# B&R Automation Studio project NAINV104C00R8L515F00 (part 4)

#### Types.typ - Exported data types
```iecst
(*HermesState*)

TYPE
	eHermesState :
		(
		HermesStateNotConnected,
		HermesStateConnected,
		HermesStateServiceDescription,
		HermesStateSServiceDescription,
		HermesStateNotAvailableNotReady,
		HermesStateBoardAvailable,
		HermesStateMachineReady,
		HermesStateAvailableAndReady,
		HermesStateTransporting,
		HermesStateTransportStopped,
		HermesStateTransportFinished
		);
END_TYPE

(**)
(*Hermes Message Type*)

TYPE
	tyHermesMsgType : 	STRUCT
		bCheckAlive : BOOL; (*Check Alive*)
		bCheckAlivePing : BOOL; (*Check Alive Ping*)
		bCheckAlivePong : BOOL; (*Check Alive Pong*)
		bServiceDescription : BOOL; (*Service Description*)
		bSServiceDescription : BOOL; (*Supervisory Service Description*)
		bNotification : BOOL; (*Notification*)
		bBoardAvailable : BOOL; (*Board Available*)
		bRevokeBoardAvailable : BOOL; (*Revoke Board Available*)
		bMachineReady : BOOL; (*Machine Ready*)
		bRevokeMachineReady : BOOL; (*Revoke Machine Ready*)
		bStartTransport : BOOL; (*Start Transport*)
		bStopTransport : BOOL; (*Stop Transport*)
		bTransportFinished : BOOL; (*Transport Finished*)
		bSetConfiguration : BOOL; (*Set Configuration*)
		bGetConfiguration : BOOL; (*Get Configuration*)
		bCurrentConfiguration : BOOL; (*Current Configuration*)
		bBoardForecast : BOOL; (*Board Forecast*)
		bBoardArrived : BOOL; (*Board Arrived*)
		bBoardDeparted : BOOL; (*Board Departed*)
		bQueryBoardInfo : BOOL; (*Query Board Info*)
		bSendBoardInfo : BOOL; (*Send Board Info*)
		bQueryWorkOrderInfo : BOOL; (*Query Work Order*)
		bSendWorkOrderInfo : BOOL; (*Send Work Order*)
		bCommand : BOOL;
	END_STRUCT;
	eHermesMsgType :
		(
		HermesMsgTypeNA, (*NA*)
		HermesMsgTypeCheckAlive, (*Check Alive*)
		HermesMsgTypeCheckAlivePing, (*Check Alive Ping*)
		HermesMsgTypeCheckAlivePong, (*Check Alive Pong*)
		HermesMsgTypeServiceDescription, (*Service Description*)
		HermesMsgTypeSServiceDescription, (*Supervisory Service Description*)
		HermesMsgTypeNotification, (*Notification*)
		HermesMsgTypeBoardAvailable, (*Board Available*)
		HermesMsgTypeRevokeBoardAvl, (*Revoke Board Available*)
		HermesMsgTypeMachineReady, (*Machine Ready*)
		HermesMsgTypeRevokeMachineReady, (*Revoke Machine Ready*)
		HermesMsgTypeStartTransport, (*Start Transport*)
		HermesMsgTypeStopTransport, (*Stop Transport*)
		HermesMsgTypeTransportFinished, (*Transport Finished*)
		HermesMsgTypeSetConfiguration, (*Set Configuration*)
		HermesMsgTypeGetConfiguration, (*Get Configuration*)
		HermesMsgTypeCurrConfiguration, (*Current Configuration*)
		HermesMsgTypeBoardForecast, (*Board Forecast*)
		HermesMsgTypeBoardForecastId, (*Board Forecast with Id*)
		HermesMsgTypeBoardForecastNoId, (*Board Forecast with no Id*)
		HermesMsgTypeBoardArrived, (*Board Arrived*)
		HermesMsgTypeBoardDeparted, (*Board Departed*)
		HermesMsgTypeQueryBoardInfo, (*Query Board Info*)
		HermesMsgTypeSendBoardInfo, (*Send Board Info*)
		HermesMsgTypeQueryWorkOrderInfo, (*Query Work Order Info*)
		HermesMsgTypeSendWorkOrderInfo, (*Send Work Order Info*)
		HermesMsgTypeCommand
		);
END_TYPE

(**)

TYPE
	eHermesCheckAliveType :
		(
		HermesCheckAliveTypeUnknown := 0, (*CheckAlive unknown*)
		HermesCheckAliveTypePing := 1, (*CheckAlive request*)
		HermesCheckAliveTypePong := 2 (*CheckAlive response*)
		);
	eHermesBoardTransfer :
		(
		HermesTransferred := 1, (*Transferred from upstream*)
		HermesLoaded := 2, (*Loaded from Magazine or a stack of Boards*)
		HermesInserted := 3 (*Inserted*)
		);
	eHermesFailedBoard :
		(
		HermesUnknownBoard := 0, (*Board of unknown quality available / Ready to accept any board*)
		HermesGoodBoard := 1, (*Good board available / Ready to accept good boards*)
		HermesFailedBoard := 2 (*Failed board available / Ready to accept failed boards*)
		);
	eHermesFlippedBoard :
		(
		HermesFlippedBoardUnknownSide := 0, (*Side up is unknown*)
		HermesFlippedBoardTopSideUp := 1, (*Board top side is up*)
		HermesFlippedBoardBtmSideUp := 2 (*Board bottom side is up*)
		);
	eHermesSeverity :
		(
		HermesSeverityFatalError := 1, (*Fatal Error*)
		HermesSeverityError := 2, (*Error*)
		HermesSeverityWarning := 3, (*Warning*)
		HermesSeverityInfo := 4 (*Info*)
		);
	eHermesTransferState :
		(
		HermesTransferStateNotStarted := 1, (*The PCB never left and hence is fully inside the upstream machine*)
		HermesTransferStateIncomplete := 2, (*The transfer was cancelled in progress*)
		HermesTransferStateComplete := 3 (*The transfer ended successfully*)
		);
END_TYPE

(**)
(**)
(*Command*)

TYPE
	tyHermesCmdProcessList : 	STRUCT
		bUSTrueDSFalse : BOOL;
		udiInterfaceString : UDINT;
		udiComMode : UDINT;
		udiCommandParam : UDINT;
	END_STRUCT;
	tyHermesCommandParam : 	STRUCT
		usiCommandIdx : USINT;
		eCommand : eHermesCommand;
		udiMsgCmdBffr : UDINT;
		a_eCommandSndQ : ARRAY[0..20]OF eHermesCommand;
	END_STRUCT;
	eHermesCommand :
		(
		HermesCommandUndefined := 0,
		HermesCommandLockInputConveyor := 1,
		HermesCommandUnLockInputConveyor := 2,
		HermesCommandRequestPause := 3,
		HermesCommandConfirmPause := 4,
		HermesCommandResumeOperation := 5,
		HermesCommandOvenInfeed := 1000,
		HermesCommandSelfDefine := 1001
		);
	tyHermesCommandPause : 	STRUCT
		bFeatureRequestTo : BOOL;
		bUnlockCoverSigTo : BOOL;
		bPrevUnlockCoverSigTo : BOOL;
		bMachineSafetySigFrom : BOOL;
		bFeatureRequestFrom : BOOL;
		bUnlockCoverSigFrom : BOOL;
		bMachineSafetySigTo : BOOL;
		bPrevMachineSafetySigTo : BOOL;
	END_STRUCT;
	tyHermesCommandLockConv : 	STRUCT
		bFeatureLockConvFrom : BOOL;
		bOvenInfoFrom : BOOL;
		bFeatureLockConvTo : BOOL;
		bOvenInfoTo : BOOL;
		bPrevOvenInfoTo : BOOL;
	END_STRUCT;
	tyHermesCommandOvenInfeed : 	STRUCT
		bFeatureOvenInfeedFrom : BOOL;
		bOvenInfeedFrom : BOOL;
		bFeatureOvenInfeedTo : BOOL;
		bOvenInfeedTo : BOOL;
		bPrevOvenInfeedTo : BOOL;
	END_STRUCT;
END_TYPE

(**)
(*Hermes Message Full Data*)

TYPE
	tyHermesNotification : 	STRUCT
		tyData : tyHermesNotificationData; (*Data*)
		tyAvl : tyHermesNotificationAvl; (*Availability*)
	END_STRUCT;
	tyHermesServiceDescription : 	STRUCT
		tyData : tyHermesServiceDescriptionData; (*Data*)
		tyAvl : tyHermesServiceDescriptionAvl; (*Availability*)
	END_STRUCT;
	tyHermesSServiceDescription : 	STRUCT
		tyData : tyHermesSServiceDescriptionData; (*Data*)
		tyAvl : tyHermesSServiceDescriptionAvl; (*Availability*)
	END_STRUCT;
	tyHermesCheckAlive : 	STRUCT
		tyData : tyHermesCheckAliveData; (*Data*)
		tyAvl : tyHermesCheckAliveAvl; (*Availability*)
	END_STRUCT;
	tyHermesBoardAvailable : 	STRUCT
		tyData : tyHermesBoardAvailableData; (*Data*)
		tyAvl : tyHermesBoardAvailableAvl; (*Availability*)
	END_STRUCT;
	tyHermesMachineReady : 	STRUCT
		tyData : tyHermesMachineReadyData; (*Data*)
		tyAvl : tyHermesMachineReadyAvl; (*Availability*)
	END_STRUCT;
	tyHermesStartTransport : 	STRUCT
		tyData : tyHermesStartTransportData; (*Data*)
		tyAvl : tyHermesStartTransportAvl; (*Availability*)
	END_STRUCT;
	tyHermesStopTransport : 	STRUCT
		tyData : tyHermesStopTransportData; (*Data*)
		tyAvl : tyHermesStopTransportAvl; (*Availability*)
	END_STRUCT;
	tyHermesTransportFinished : 	STRUCT
		tyData : tyHermesTransportFinishedData; (*Data*)
		tyAvl : tyHermesTransportFinishedAvl; (*Availability*)
	END_STRUCT;
	tyHermesBoardForecast : 	STRUCT
		tyData : tyHermesBoardForecastData; (*Data*)
		tyAvl : tyHermesBoardForecastAvl; (*Availability*)
	END_STRUCT;
	tyHermesQueryBoardInfo : 	STRUCT
		tyData : tyHermesQueryBoardInfoData; (*Data*)
		tyAvl : tyHermesQueryBoardInfoAvl; (*Availability*)
	END_STRUCT;
	tyHermesSendBoardInfo : 	STRUCT
		tyData : tyHermesSendBoardInfoData; (*Data*)
		tyAvl : tyHermesSendBoardInfoAvl; (*Availability*)
	END_STRUCT;
	tyHermesBoardArrived : 	STRUCT
		tyData : tyHermesBoardArrivedData; (*Data*)
		tyAvl : tyHermesBoardArrivedAvl; (*Availability*)
	END_STRUCT;
	tyHermesBoardDeparted : 	STRUCT
		tyData : tyHermesBoardDepartedData; (*Data*)
		tyAvl : tyHermesBoardDepartedAvl; (*Availability*)
	END_STRUCT;
	tyHermesSetConfiguration : 	STRUCT
		tyData : tyHermesSetConfigurationData; (*Data*)
		tyAvl : tyHermesSetConfigurationAvl; (*Availability*)
	END_STRUCT;
	tyHermesCurrentConfiguration : 	STRUCT
		tyData : tyHermesCurrentConfigurationData; (*Data*)
		tyAvl : tyHermesCurrentConfigurationAvl; (*Availability*)
	END_STRUCT;
	tyHermesQueryWorkOrderInfo : 	STRUCT
		tyData : tyHermesQueryWorkOrderInfoData; (*Data*)
		tyAvl : tyHermesQueryWorkOrderInfoAvl; (*Availability*)
	END_STRUCT;
	tyHermesSendWorkOrderInfo : 	STRUCT
		tyData : tyHermesSendWorkOrderInfoData; (*Data*)
		tyAvl : tyHermesSendWorkOrderInfoAvl; (*Availability*)
	END_STRUCT;
	tyHermesCommand : 	STRUCT
		tyData : tyHermesCommandData; (*Data*)
		tyAvl : tyHermesCommandAvl; (*Availability*)
	END_STRUCT;
END_TYPE

(**)
(*Hermes Message Data*)

TYPE
	tyHermesNotificationData : 	STRUCT
		iNotificationCode : INT; (*A notification code of the list below. Notification codes above 1000 are not defined by this protocol and may be used by the application.*)
		eSeverity : eHermesSeverity; (*Notification Severity*)
		sDescription : STRING[254]; (*An English textual description of the notification.*)
	END_STRUCT;
	tyHermesServiceDescriptionData : 	STRUCT
		sMachineId : STRING[80]; (*ID/name of the sending machine for identifying it in a Hermes enabled production line.*)
		sSystemId : STRING[80]; (*ID / name of the sending machine or supervisory system for identifying it in a Hermes enabled production line. 	*)
		iLaneId : INT; (*The sending machine's lane to which this connection is relating to. Lanes are enumerated looking downstream from right to left beginning with 1.*)
		sInterfaceId : STRING[80]; (*The ID of the sending machine's transportation interface to which this connection is relating to.*)
		sVersion : STRING[7]; (*The implemented interface version of the machine.*)
		tySupportedFeatures : tyHermesFeature; (*List of supported features (empty for version 1.0)*)
	END_STRUCT;
	tyHermesSServiceDescriptionData : 	STRUCT
		sSystemId : STRING[80]; (*ID / name of the sending machine or supervisory system for identifying it in a Hermes enabled production line. 	*)
		sMachineId : STRING[80]; (*ID/name of the sending machine for identifying it in a Hermes enabled production line.*)
		sVersion : STRING[7]; (*The implemented interface version of the machine.*)
		tySupportedFeatures : tyHermesSvyFeature; (*List of supported features (empty for version 1.0)*)
	END_STRUCT;
	tyHermesFeature : 	STRUCT
		bFeatureCheckAliveResponse : BOOL; (*Indication of CheckAliveResponse function implementation.*)
		bFeatureBoardForecast : BOOL; (*Indication of BoardForecastfunction implementation.*)
		bFeatureConfiguration : BOOL; (*Indication of Configuration function implementation.*)
		bFeatureBoardTracking : BOOL; (*Indication of BoardTracking function implementation.*)
		bFeatureQueryWorkOrderInfo : BOOL; (*Indication of QueryWorkOrderInfo function implementation.*)
		bFeatureSendWorkOrderInfo : BOOL; (*Indication of SendWorkOrderInfo function implementation.*)
		bFeatureQueryBoardInfo : BOOL; (*Indication of QueryBoardInfo function implementation.*)
		bFeatureSendBoardInfo : BOOL; (*Indication of SendBoardInfo function implementation.*)
		bFeatureCommand : BOOL; (*Indication of SendBoardInfo function implementation.*)
	END_STRUCT;
	tyHermesSvyFeature : 	STRUCT
		bFeatureCheckAliveResponse : BOOL; (*Indication of CheckAliveResponse function implementation.*)
		bFeatureConfiguration : BOOL; (*Indication of Configuration  function implementation.*)
		bFeatureBoardTracking : BOOL; (*Indication of BoardTracking function implementation.*)
		bFeatureQueryWorkOrderInfo : BOOL; (*Indication of QueryWorkOrderInfo function implementation.*)
		bFeatureSendWorkOrderInfo : BOOL; (*Indication of SendWorkOrderInfo function implementation.*)
	END_STRUCT;
	tyHermesCheckAliveData : 	STRUCT
		eType : eHermesCheckAliveType; (*Ping / Pong message type*)
		sId : STRING[80]; (*Identifier of the message*)
	END_STRUCT;
	tyHermesBoardAvailableData : 	STRUCT
		sBoardId : STRING[36]; (*Indicating the ID of the available board*)
		sBoardIdCreatedBy : STRING[80]; (*MachineId of the machine which created the BoardId (the first machine in a consecutive row of machines implementing this protocol). The MachineId is part of the Hermes Configuration.*)
		eFailedBoard : eHermesFailedBoard; (*A value of Unknown Board, Good Board & Failed Board*)
		sProductTypeId : STRING[254]; (*Identifies a collection of PCBs sharing common properties.*)
		eFlippedBoard : eHermesFlippedBoard; (*A value of Unknown Side, Top Side Up & Bottom Side Up.*)
		sTopBarcode : STRING[254]; (*The barcode of the top side of the PCB*)
		sBottomBarcode : STRING[254]; (*The barcode of the bottom side of the PCB*)
		rLength : REAL; (*The length of the PCB in millimeter.*)
		rWidth : REAL; (*The width of the PCB in millimeter.*)
		rThickness : REAL; (*The thickness of the PCB in millimeter.*)
		rConveyorSpeed : REAL; (*The conveyor speed preferred by the upstream machine in millimeter per second.*)
		rTopClearanceHeight : REAL; (*The clearance height for the top side of the PCB in millimeter.*)
		rBottomClearanceHeight : REAL; (*The clearance height for the bottom side of the PCB in millimeter.*)
		rWeight : REAL; (*The weight of the PCB in grams.*)
		sWorkOrderId : STRING[80]; (*The work order for the production of PCB.*)
		sBatchId : STRING[80]; (*The batch id of a splitted work order.*)
		iRoute : INT; (*The routing instuction to DS machine*)
		iAction : INT; (*The action instuction to DS machine (mode change)*)
		tySubBoards : tyHermesBASubBoardsData;
	END_STRUCT;
	tyHermesBASubBoardsData : 	STRUCT
		iSubBoardsPos : ARRAY[0..4]OF INT; (*A value of Unknown Board, Good Board & Failed Board*)
		sSubBoardsBc : ARRAY[0..4]OF STRING[80]; (*If responding to a BoardForecast message mandatory. It indicates the ID of the original BoardForecast message.*)
		iSubBoardsSt : ARRAY[0..4]OF INT; (*Indicating the ID of the board that will be handed over as next. In case of product change this attribute will not be sent.*)
	END_STRUCT;
	tyHermesMachineReadyData : 	STRUCT
		eFailedBoard : eHermesFailedBoard; (*A value of Unknown Board, Good Board & Failed Board*)
		sForecastId : STRING[80]; (*If responding to a BoardForecast message mandatory. It indicates the ID of the original BoardForecast message.*)
		sBoardId : STRING[36]; (*Indicating the ID of the board that will be handed over as next. In case of product change this attribute will not be sent.*)
		sProductTypeId : STRING[254]; (*Identifies a collection of PCBs sharing common properties.*)
		eFlippedBoard : eHermesFlippedBoard; (*A value of Unknown Side, Top Side Up & Bottom Side Up.*)
		rLength : REAL; (*The length of the PCB in millimeter.*)
		rWidth : REAL; (*The width of the PCB in millimeter.*)
		rThickness : REAL; (*The thickness of the PCB in millimeter.*)
		rConveyorSpeed : REAL; (*The conveyor speed preferred by the upstream machine in millimeter per second.*)
		rTopClearanceHeight : REAL; (*The clearance height for the top side of the PCB in millimeter.*)
		rBottomClearanceHeight : REAL; (*The clearance height for the bottom side of the PCB in millimeter.*)
		rWeight : REAL; (*The weight of the PCB in grams.*)
		sWorkOrderId : STRING[80]; (*The work order for the production of PCB.*)
		sBatchId : STRING[80]; (*The batch id of a splitted work order.*)
	END_STRUCT;
	tyHermesStartTransportData : 	STRUCT
		sBoardId : STRING[36]; (*The ID of the board for which the transport shall be started.*)
		rConveyorSpeed : REAL; (*Optional parameter indicating the selected conveyor speed for the handover in millimeter per second.*)
	END_STRUCT;
	tyHermesStopTransportData : 	STRUCT
		eTransferState : eHermesTransferState; (*Transfer States*)
		sBoardId : STRING[36]; (*The ID of the board to which the message relates to.*)
	END_STRUCT;
	tyHermesTransportFinishedData : 	STRUCT
		eTransferState : eHermesTransferState; (*Transfer States*)
		sBoardId : STRING[36]; (*The ID of the board to which the message relates to.*)
	END_STRUCT;
	tyHermesBoardForecastData : 	STRUCT
		sForecastId : STRING[80]; (*Indicating the ID of forecast message. The ID must be unambiguous and e.g. can be a timetamp or a GUID.*)
		rTimeUntilAvailable : REAL; (*Number of seconds until a board may be available at downstream machine.*)
		sBoardId : STRING[36]; (*Indicating the ID of the board that will be handed over as next. In case of product change this field will not be sent.*)
		sBoardIdCreatedBy : STRING[80]; (*MachineId of the machine which created the BoardId*)
		eFailedBoard : eHermesFailedBoard; (*A value of Unknown Board, Good Board & Failed Board*)
		sProductTypeId : STRING[254]; (*Identifies a collection of PCBs sharing common properties.*)
		eFlippedBoard : eHermesFlippedBoard; (*A value of Unknown Side, Top Side Up & Bottom Side Up.*)
		sTopBarcode : STRING[254]; (*The barcode of the top side of the next PCB*)
		sBottomBarcode : STRING[254]; (*The barcode of the bottom side of the next PCB*)
		rLength : REAL; (*The length of the PCB in millimeter.*)
		rWidth : REAL; (*The width of the PCB in millimeter.*)
		rThickness : REAL; (*The thickness of the PCB in millimeter.*)
		rConveyorSpeed : REAL; (*The conveyor speed preferred by the upstream machine in millimeter per second.*)
		rTopClearanceHeight : REAL; (*The clearance height for the top side of the PCB in millimeter.*)
		rBottomClearanceHeight : REAL; (*The clearance height for the bottom side of the PCB in millimeter.*)
		rWeight : REAL; (*The weight of the PCB in grams.*)
		sWorkOrderId : STRING[80]; (*The work order for the production of PCB.*)
		sBatchId : STRING[80]; (*The batch id of a splitted work order.*)
	END_STRUCT;
	tyHermesQueryBoardInfoData : 	STRUCT
		sTopBarcode : STRING[254]; (*The barcode of the top side of the PCB. Either top or bottom barcode must be specified.*)
		sBottomBarcode : STRING[254]; (*The barcode of the bottom side of the PCB. Either top or bottom barcode must be specified.*)
	END_STRUCT;
	tyHermesSendBoardInfoData : 	STRUCT
		sBoardId : STRING[36]; (*The ID of the board which data has been requested. This attribute will not be sent if the board information has not been found.*)
		sBoardIdCreatedBy : STRING[80]; (*MachineId of the machine which created the BoardId. This attribute will not be sent if the board information has not been found.*)
		eFailedBoard : eHermesFailedBoard; (*A value of Unknown Board, Good Board & Failed Board. This attribute will not be sent if the board information has not been found.*)
		sProductTypeId : STRING[254]; (*Identifies a collection of PCBs sharing common properties.*)
		eFlippedBoard : eHermesFlippedBoard; (*A value of Unknown Side, Top Side Up & Bottom Side Up. This attribute will not be sent if the board information has not been found.*)
		sTopBarcode : STRING[254]; (*The barcode of the top side of the next PCB. This attribute is mandatory if it has been in the QueryBoardInfo message.*)
		sBottomBarcode : STRING[254]; (*The barcode of the bottom side of the next PCB. This attribute is mandatory if it has been in the QueryBoardInfo message.*)
		rLength : REAL; (*The length of the PCB in millimeter.*)
		rWidth : REAL; (*The width of the PCB in millimeter.*)
		rThickness : REAL; (*The thickness of the PCB in millimeter.*)
		rTopClearanceHeight : REAL; (*The clearance height for the top side of the PCB in millimeter.*)
		rBottomClearanceHeight : REAL; (*The clearance height for the bottom side of the PCB in millimeter.*)
		rWeight : REAL; (*The weight of the PCB in grams.*)
		sWorkOrderId : STRING[80]; (*The work order for the production of PCB.*)
		sBatchId : STRING[80]; (*The batch id of a splitted work order.*)
	END_STRUCT;
	tyHermesBoardArrivedData : 	STRUCT
		sMachineId : STRING[80]; (*ID / name of this machine for identifying it in a Hermes enabled production line. 	*)
		iUpstreamLaneId : INT; (*The lane on the upstream side. Lanes are enumerated looking downstream from right to left beginning with 1.*)
		sUpstreamInterfaceId : STRING[80]; (*The ID of the transportation interface on the upstream side.*)
		sMagazineId : STRING[80]; (*Barcode of a magazine, required to identify the magazine from which the Board was transferred.*)
		iSlotId : INT; (*Indicates the slot in the magazine, enumerated from bottom to top, beginning with 1.*)
		eBoadTransfer : eHermesBoardTransfer; (*A value of BoardTransferred or Board Loaded or Board Inserted.*)
		sBoardId : STRING[36]; (*Indicating the ID of the available board. 	*)
		sBoardIdCreatedBy : STRING[80]; (*MachineId of the machine which created the BoardId (the first machine in a consecutive row of machines implementing this protocol). The MachineId is part of the Hermes configuration.*)
		eFailedBoard : eHermesFailedBoard; (*A value of Unknown Board, Good Board & Failed Board*)
		sProductTypeId : STRING[254]; (*Identifies a collection of PCBs sharing common properties.*)
		eFlippedBoard : eHermesFlippedBoard; (*A value of Unknown Side, Top Side Up & Bottom Side Up.*)
		sTopBarcode : STRING[254]; (*The barcode of the top side of the next PCB*)
		sBottomBarcode : STRING[254]; (*The barcode of the bottom side of the next PCB*)
		rLength : REAL; (*The length of the PCB in millimeter.*)
		rWidth : REAL; (*The width of the PCB in millimeter.*)
		rThickness : REAL; (*The thickness of the PCB in millimeter.*)
		rConveyorSpeed : REAL; (*The conveyor speed preferred by the upstream machine in millimeter per second.*)
		rTopClearanceHeight : REAL; (*The clearance height for the top side of the PCB in millimeter.*)
		rBottomClearanceHeight : REAL; (*The clearance height for the bottom side of the PCB in millimeter.*)
		rWeight : REAL; (*The weight of the PCB in grams.*)
		sWorkOrdedId : STRING[80]; (*The work order for the production of PCB.*)
		sBatchId : STRING[80]; (*The batch id of a splitted work order.*)
		iRoute : INT;
		iAction : INT;
	END_STRUCT;
	tyHermesBoardDepartedData : 	STRUCT
		sMachineId : STRING[80]; (*ID / name of this machine for identifying it in a Hermes enabled production line. 	*)
		iDownstreamLaneId : INT; (*The lane on the downstream side. Lanes are enumerated looking downstream from right to left beginning with 1.*)
		sDownstreamInterfaceId : STRING[80]; (*The ID of the transportation interface on the downstream side.*)
		sMagazineId : STRING[80]; (*Barcode of a magazine, required to identify the magazine from which the Board was transferred.*)
		iSlotId : INT; (*Indicates the slot in the magazine, enumerated from bottom to top, beginning with 1.*)
		eBoadTransfer : eHermesBoardTransfer; (*A value of BoardTransferred or Board Loaded or Board Inserted.*)
		sBoardId : STRING[36]; (*Indicating the ID of the available board. 	*)
		sBoardIdCreatedBy : STRING[80]; (*MachineId of the machine which created the BoardId (the first machine in a consecutive row of machines implementing this protocol). The MachineId is part of the Hermes configuration.*)
		eFailedBoard : eHermesFailedBoard; (*A value of Unknown Board, Good Board & Failed Board*)
		sProductTypeId : STRING[254]; (*Identifies a collection of PCBs sharing common properties.*)
		eFlippedBoard : eHermesFlippedBoard; (*A value of Unknown Side, Top Side Up & Bottom Side Up.*)
		sTopBarcode : STRING[254]; (*The barcode of the top side of the next PCB*)
		sBottomBarcode : STRING[254]; (*The barcode of the bottom side of the next PCB*)
		rLength : REAL; (*The length of the PCB in millimeter.*)
		rWidth : REAL; (*The width of the PCB in millimeter.*)
		rThickness : REAL; (*The thickness of the PCB in millimeter.*)
		rConveyorSpeed : REAL; (*The conveyor speed preferred by the upstream machine in millimeter per second.*)
		rTopClearanceHeight : REAL; (*The clearance height for the top side of the PCB in millimeter.*)
		rBottomClearanceHeight : REAL; (*The clearance height for the bottom side of the PCB in millimeter.*)
		rWeight : REAL; (*The weight of the PCB in grams.*)
		sWorkOrdedId : STRING[80]; (*The work order for the production of PCB.*)
		sBatchId : STRING[80]; (*The batch id of a splitted work order.*)
		iRoute : INT;
		iAction : INT;
	END_STRUCT;
	tyHermesQueryWorkOrderInfoData : 	STRUCT
		sQueryId : STRING[80]; (*Indicates the ID of QueryWorkOrder message. The ID must be unambiguous and e.g. can be a timestamp or a GUID.*)
		sMachineId : STRING[80]; (*ID / name of this machine for identifying it in a Hermes enabled production line.*)
		sMagazineId : STRING[80]; (*Barcode of a magazine, required to identify the magazine.*)
		iSlotId : INT; (*Indicates the slot in the magazine, enumerated from bottom to top, beginning with 1.*)
		sBarcode : STRING[254]; (*The barcode of the PCB.*)
	END_STRUCT;
	tyHermesSendWorkOrderInfoData : 	STRUCT
		sQueryId : STRING[80]; (*ID of QueryWorkOrderInfo this message refers to. This attribute is mandatory if it has been in the QueryWorkOrderInfo message.*)
		sWorkOrderId : STRING[80]; (*Identifies the work order for production of the PCB.*)
		sBatchId : STRING[80]; (*The batch id of a splitted work order.*)
		sBoardId : STRING[36]; (*Indicating the ID of the available board.*)
		sBoardIdCreatedBy : STRING[80]; (*MachineId of the machine which created the BoardId (the first machine in a consecutive row of machines implementing this protocol). The MachineId is part of the Hermes configuration.*)
		eFailedBoard : eHermesFailedBoard; (*A value of Unknown Board, Good Board & Failed Board. This attribute will not be sent if the board information has not been found.*)
		sProductTypeId : STRING[254]; (*Identifies a collection of PCBs sharing common properties.*)
		eFlippedBoard : eHermesFlippedBoard; (*A value of Unknown Side, Top Side Up & Bottom Side Up. This attribute will not be sent if the board information has not been found.*)
		sTopBarcode : STRING[254]; (*The barcode of the top side of the next PCB. This attribute is mandatory if it has been in the QueryBoardInfo message.*)
		sBottomBarcode : STRING[254]; (*The barcode of the bottom side of the next PCB. This attribute is mandatory if it has been in the QueryBoardInfo message.*)
		rLength : REAL; (*The length of the PCB in millimeter.*)
		rWidth : REAL; (*The width of the PCB in millimeter.*)
		rThickness : REAL; (*The thickness of the PCB in millimeter.*)
		rConveyorSpeed : REAL; (*The thickness of the PCB in millimeter.*)
		rTopClearanceHeight : REAL; (*The clearance height for the top side of the PCB in millimeter.*)
		rBottomClearanceHeight : REAL; (*The clearance height for the bottom side of the PCB in millimeter.*)
		rWeight : REAL; (*The weight of the PCB in grams.*)
		iRoute : INT;
	END_STRUCT;
	tyHermesCommandData : 	STRUCT
		eCommand : eHermesCommand;
	END_STRUCT;
	tyHermesSetConfigurationData : 	STRUCT
		sMachineId : STRING[80]; (*ID/name of this machine for identifying it in a Hermes enabled production line*)
		uiSupervisorySystemPort : UINT; (*Supervisory system port number.*)
		a_tyUpstreamConfigurations : ARRAY[0..c_diHermesConfigMaxIdx]OF tyHermesUpstreamConfiguration; (*Configuration for upstream lanes*)
		a_tyDownstreamConfigurations : ARRAY[0..c_diHermesConfigMaxIdx]OF tyHermesDownstreamConfiguration; (*Configuration for downstream lanes*)
	END_STRUCT;
	tyHermesCurrentConfigurationData : 	STRUCT
		sMachineId : STRING[80]; (*ID/name of this machine for identifying it in a Hermes enabled production line*)
		uiSupervisorySystemPort : UINT; (*Supervisory system port number.*)
		a_tyUpstreamConfigurations : ARRAY[0..c_diHermesConfigMaxIdx]OF tyHermesUpstreamConfiguration; (*Configuration for upstream lanes*)
		a_tyDownstreamConfigurations : ARRAY[0..c_diHermesConfigMaxIdx]OF tyHermesDownstreamConfiguration; (*Configuration for downstream lanes*)
	END_STRUCT;
	tyHermesUpstreamConfiguration : 	STRUCT
		iUpstreamLaneId : INT; (*The lane on the upstream side Lanes are enumerated looking downstream from right to left beginning with 1*)
		sUpstreamInterfaceId : STRING[80]; (*The ID of the transportation interface on the upstream side*)
		sHostAddress : STRING[254]; (*The IP address or hostname of the upstream machine for this lane and transportation interface*)
		uiPort : UINT; (*Port number on which connections shall be established*)
	END_STRUCT;
	tyHermesDownstreamConfiguration : 	STRUCT
		iDownstreamLaneId : INT; (*The lane on the downstream side Lanes are enumerated looking downstream from right to left beginning with 1*)
		sDownstreamInterfaceId : STRING[80]; (*The ID of the transportation interface on the downstream side*)
		sClientAddress : STRING[254]; (*The IP address or hostname of the downstream machine for this lane and transportation interface. If not specified, then connections from any IP address are accepted.*)
		uiPort : UINT; (*Port number on which the server shall accept connections for this lane*)
	END_STRUCT;
END_TYPE

(**)
(*Hermes Message Data Availability*)

TYPE
	tyHermesNotificationAvl : 	STRUCT
		bNotificationCode : BOOL; (*A notification code of the list below. Notification codes above 1000 are not defined by this protocol and may be used by the application.*)
		bSeverity : BOOL; (*Notification Severity*)
		bDescription : BOOL; (*An English textual description of the notification.*)
	END_STRUCT;
	tyHermesServiceDescriptionAvl : 	STRUCT
		bMachineId : BOOL; (*ID/name of the sending machine for identifying it in a Hermes enabled production line.*)
		bSystemId : BOOL; (*ID / name of the sending machine or supervisory system for identifying it in a Hermes enabled production line. 	*)
		bLaneId : BOOL; (*The sending machine's lane to which this connection is relating to. Lanes are enumerated looking downstream from right to left beginning with 1.*)
		bInterfaceId : BOOL; (*The ID of the sending machine's transportation interface to which this connection is relating to.*)
		bVersion : BOOL; (*The implemented interface version of the machine.*)
		bSupportedFeatures : BOOL; (*List of supported features (empty for version 1.0)*)
		tySupportedFeatures : tyHermesFeatureAvl; (*List of supported features (empty for version 1.0)*)
	END_STRUCT;
	tyHermesSServiceDescriptionAvl : 	STRUCT
		bSystemId : BOOL; (*ID / name of the sending machine or supervisory system for identifying it in a Hermes enabled production line. 	*)
		bMachineId : BOOL; (*ID/name of the sending machine for identifying it in a Hermes enabled production line.*)
		bVersion : BOOL; (*The implemented interface version of the machine.*)
		bSupportedFeatures : BOOL; (*List of supported features (empty for version 1.0)*)
		tySupportedFeatures : tyHermesSvyFeatureAvl; (*List of supported features (empty for version 1.0)*)
	END_STRUCT;
	tyHermesFeatureAvl : 	STRUCT
		bFeatureCheckAliveResponse : BOOL; (*Indication of CheckAliveResponse function implementation.*)
		bFeatureBoardForecast : BOOL; (*In the upstream role: Machine emits BoardForecast messages.*)
		bFeatureQueryBoardInfo : BOOL; (*Indication of QueryBoardInfo function implementation.*)
		bFeatureSendBoardInfo : BOOL; (*Indication of SendBoardInfo function implementation.*)
		bFeatureCommand : BOOL;
	END_STRUCT;
	tyHermesSvyFeatureAvl : 	STRUCT
		bFeatureConfiguration : BOOL; (*Indication of configuration functions implementation.*)
		bFeatureCheckAliveResponse : BOOL; (*Indication of CheckAliveResponse function implementation.*)
		bFeatureBoardTracking : BOOL; (*Indication of board tracking functions implementation.*)
		bFeatureQueryWorkOrderInfo : BOOL; (*Indication of QueryWorkOrderInfo function implementation.*)
		bFeatureSendWorkOrderInfo : BOOL; (*Indication of SendWorkOrderInfo function implementation.*)
	END_STRUCT;
	tyHermesCheckAliveAvl : 	STRUCT
		bType : BOOL; (*Ping / Pong message type*)
		bId : BOOL; (*Identifier of the message*)
	END_STRUCT;
	tyHermesBoardAvailableAvl : 	STRUCT
		bBoardId : BOOL; (*Indicating the ID of the available board*)
		bBoardIdCreatedBy : BOOL; (*MachineId of the machine which created the BoardId (the first machine in a consecutive row of machines implementing this protocol). The MachineId is part of the Hermes configuration.*)
		bFailedBoard : BOOL; (*A value of Unknown Board, Good Board & Failed Board*)
		bProductTypeId : BOOL; (*Identifies a collection of PCBs sharing common properties.*)
		bFlippedBoard : BOOL; (*A value of Unknown Side, Top Side Up & Bottom Side Up.*)
		bTopBarcode : BOOL; (*The barcode of the top side of the PCB*)
		bBottomBarcode : BOOL; (*The barcode of the bottom side of the PCB*)
		bLength : BOOL; (*The length of the PCB in millimeter.*)
		bWidth : BOOL; (*The width of the PCB in millimeter.*)
		bThickness : BOOL; (*The thickness of the PCB in millimeter.*)
		bConveyorSpeed : BOOL; (*The conveyor speed preferred by the upstream machine in millimeter per second.*)
		bTopClearanceHeight : BOOL; (*The clearance height for the top side of the PCB in millimeter.*)
		bBottomClearanceHeight : BOOL; (*The clearance height for the bottom side of the PCB in millimeter.*)
		bWeight : BOOL; (*The weight of the PCB in grams.*)
		bWorkOrderId : BOOL; (*The work order for the production of PCB.*)
		bBatchId : BOOL; (*The batch id of a splitted work order.*)
		bRoute : BOOL;
		bAction : BOOL;
		tySubBoards : tyHermesBASubBoardsAvl;
	END_STRUCT;
	tyHermesBASubBoardsAvl : 	STRUCT
		bSubBoardsPos : ARRAY[0..4]OF BOOL; (*A value of Unknown Board, Good Board & Failed Board*)
		bSubBoardsBc : ARRAY[0..4]OF BOOL; (*If responding to a BoardForecast message mandatory. It indicates the ID of the original BoardForecast message.*)
		bSubBoardsSt : ARRAY[0..4]OF BOOL; (*Indicating the ID of the board that will be handed over as next. In case of product change this attribute will not be sent.*)
	END_STRUCT;
	tyHermesMachineReadyAvl : 	STRUCT
		bFailedBoard : BOOL; (*A value of Unknown Board, Good Board & Failed Board*)
		bForecastId : BOOL; (*If responding to a BoardForecast message mandatory. It indicates the ID of the original BoardForecast message.*)
		bBoardId : BOOL; (*Indicating the ID of the board that will be handed over as next. In case of product change this attribute will not be sent.*)
		bProductTypeId : BOOL; (*Identifies a collection of PCBs sharing common properties.*)
		bFlippedBoard : BOOL; (*A value of Unknown Side, Top Side Up & Bottom Side Up.*)
		bLength : BOOL; (*The length of the PCB in millimeter.*)
		bWidth : BOOL; (*The width of the PCB in millimeter.*)
		bThickness : BOOL; (*The thickness of the PCB in millimeter.*)
		bConveyorSpeed : BOOL; (*The conveyor speed preferred by the upstream machine in millimeter per second.*)
		bTopClearanceHeight : BOOL; (*The clearance height for the top side of the PCB in millimeter.*)
		bBottomClearanceHeight : BOOL; (*The clearance height for the bottom side of the PCB in millimeter.*)
		bWeight : BOOL; (*The weight of the PCB in grams.*)
		bWorkOrderId : BOOL; (*The work order for the production of PCB.*)
		bBatchId : BOOL; (*The batch id of a splitted work order.*)
	END_STRUCT;
	tyHermesStartTransportAvl : 	STRUCT
		bBoardId : BOOL; (*The ID of the board for which the transport shall be started.*)
		bConveyorSpeed : BOOL; (*Optional parameter indicating the selected conveyor speed for the handover in millimeter per second.*)
	END_STRUCT;
	tyHermesStopTransportAvl : 	STRUCT
		bTransferState : BOOL; (*Transfer States*)
		bBoardId : BOOL; (*The ID of the board to which the message relates to.*)
	END_STRUCT;
	tyHermesTransportFinishedAvl : 	STRUCT
		bTransferState : BOOL; (*Transfer States*)
		bBoardId : BOOL; (*The ID of the board to which the message relates to.*)
	END_STRUCT;
	tyHermesBoardForecastAvl : 	STRUCT
		bForecastId : BOOL; (*Indicating the ID of forecast message. The ID must be unambiguous and e.g. can be a timetamp or a GUID.*)
		bTimeUntilAvailable : BOOL; (*Number of seconds until a board may be available at downstream machine.*)
		bBoardId : BOOL; (*Indicating the ID of the board that will be handed over as next. In case of product change this field will not be sent.*)
		bBoardIdCreatedBy : BOOL; (*MachineId of the machine which created the BoardId (the first machine in a consecutive row of machines implementing this protocol). The MachineId is part of the Hermes configuration.*)
		bFailedBoard : BOOL; (*A value of Unknown Board, Good Board & Failed Board*)
		bProductTypeId : BOOL; (*Identifies a collection of PCBs sharing common properties.*)
		bFlippedBoard : BOOL; (*A value of Unknown Side, Top Side Up & Bottom Side Up.*)
		bTopBarcode : BOOL; (*The barcode of the top side of the next PCB*)
		bBottomBarcode : BOOL; (*The barcode of the bottom side of the next PCB*)
		bLength : BOOL; (*The length of the PCB in millimeter.*)
		bWidth : BOOL; (*The width of the PCB in millimeter.*)
		bThickness : BOOL; (*The thickness of the PCB in millimeter.*)
		bConveyorSpeed : BOOL; (*The conveyor speed preferred by the upstream machine in millimeter per second.*)
		bTopClearanceHeight : BOOL; (*The clearance height for the top side of the PCB in millimeter.*)
		bBottomClearanceHeight : BOOL; (*The clearance height for the bottom side of the PCB in millimeter.*)
		bWeight : BOOL; (*The weight of the PCB in grams.*)
		bWorkOrderId : BOOL; (*The work order for the production of PCB.*)
		bBatchId : BOOL; (*The batch id of a splitted work order.*)
	END_STRUCT;
	tyHermesQueryBoardInfoAvl : 	STRUCT
		bTopBarcode : BOOL; (*The barcode of the top side of the PCB. Either top or bottom barcode must be specified.*)
		bBottomBarcode : BOOL; (*The barcode of the bottom side of the PCB. Either top or bottom barcode must be specified.*)
	END_STRUCT;
	tyHermesSendBoardInfoAvl : 	STRUCT
		bBoardId : BOOL; (*The ID of the board which data has been requested. This attribute will not be sent if the board information has not been found.*)
		bBoardIdCreatedBy : BOOL; (*MachineId of the machine which created the BoardId (the first machine in a consecutive row of machines implementing this protocol). The MachineId is part of the Hermes configuration.*)
		bFailedBoard : BOOL; (*A value of Unknown Board, Good Board & Failed Board. This attribute will not be sent if the board information has not been found.*)
		bProductTypeId : BOOL; (*Identifies a collection of PCBs sharing common properties.*)
		bFlippedBoard : BOOL; (*A value of Unknown Side, Top Side Up & Bottom Side Up. This attribute will not be sent if the board information has not been found.*)
		bTopBarcode : BOOL; (*The barcode of the top side of the next PCB. This attribute is mandatory if it has been in the QueryBoardInfo message.*)
		bBottomBarcode : BOOL; (*The barcode of the bottom side of the next PCB. This attribute is mandatory if it has been in the QueryBoardInfo message.*)
		bLength : BOOL; (*The length of the PCB in millimeter.*)
		bWidth : BOOL; (*The width of the PCB in millimeter.*)
		bThickness : BOOL; (*The thickness of the PCB in millimeter.*)
		bTopClearanceHeight : BOOL; (*The clearance height for the top side of the PCB in millimeter.*)
		bBottomClearanceHeight : BOOL; (*The clearance height for the bottom side of the PCB in millimeter.*)
		bWeight : BOOL; (*The weight of the PCB in grams.*)
		bWorkOrderId : BOOL; (*The work order for the production of PCB.*)
		bBatchId : BOOL; (*The batch id of a splitted work order.*)
	END_STRUCT;
	tyHermesBoardArrivedAvl : 	STRUCT
		bMachineId : BOOL; (*ID / name of this machine for identifying it in a Hermes enabled production line. 	*)
		bUpstreamLaneId : BOOL; (*The lane on the upstream side. Lanes are enumerated looking downstream from right to left beginning with 1.*)
		bUpstreamInterfaceId : BOOL; (*The ID of the transportation interface on the upstream side.*)
		bMagazineId : BOOL; (*Barcode of a magazine, required to identify the magazine from which the Board was transferred.*)
		bSlotId : BOOL; (*Indicates the slot in the magazine, enumerated from bottom to top, beginning with 1.*)
		bBoardTransfer : BOOL; (*A value of BoardTransferred or Board Loaded or Board Inserted.*)
		bBoardId : BOOL; (*Indicating the ID of the available board. 	*)
		bBoardIdCreatedBy : BOOL; (*MachineId of the machine which created the BoardId (the first machine in a consecutive row of machines implementing this protocol). The MachineId is part of the Hermes configuration.*)
		bFailedBoard : BOOL; (*A value of Unknown Board, Good Board & Failed Board*)
		bProductTypeId : BOOL; (*Identifies a collection of PCBs sharing common properties.*)
		bFlippedBoard : BOOL; (*A value of Unknown Side, Top Side Up & Bottom Side Up.*)
		bTopBarcode : BOOL; (*The barcode of the top side of the next PCB*)
		bBottomBarcode : BOOL; (*The barcode of the bottom side of the next PCB*)
		bLength : BOOL; (*The length of the PCB in millimeter.*)
		bWidth : BOOL; (*The width of the PCB in millimeter.*)
		bThickness : BOOL; (*The thickness of the PCB in millimeter.*)
		bConveyorSpeed : BOOL; (*The conveyor speed preferred by the upstream machine in millimeter per second.*)
		bTopClearanceHeight : BOOL; (*The clearance height for the top side of the PCB in millimeter.*)
		bBottomClearanceHeight : BOOL; (*The clearance height for the bottom side of the PCB in millimeter.*)
		bWeight : BOOL; (*The weight of the PCB in grams.*)
		bWorkOrderId : BOOL; (*The work order for the production of PCB.*)
		bBatchId : BOOL; (*The batch id of a splitted work order.*)
		bRoute : BOOL;
		bAction : BOOL;
	END_STRUCT;
	tyHermesBoardDepartedAvl : 	STRUCT
		bMachineId : BOOL; (*ID / name of this machine for identifying it in a Hermes enabled production line. 	*)
		bDownstreamLaneId : BOOL; (*The lane on the downstream side. Lanes are enumerated looking downstream from right to left beginning with 1.*)
		bDownstreamInterfaceId : BOOL; (*The ID of the transportation interface on the downstream side.*)
		bMagazineId : BOOL; (*Barcode of a magazine, required to identify the magazine to which the Board was transferred.*)
		bSlotId : BOOL; (*Indicates the slot in the magazine, enumerated from bottom to top, beginning with 1.*)
		bBoardTransfer : BOOL; (*A value of BoardTransferred or Board Loaded or Board Inserted.*)
		bBoardId : BOOL; (*Indicating the ID of the available board. 	*)
		bBoardIdCreatedBy : BOOL; (*MachineId of the machine which created the BoardId (the first machine in a consecutive row of machines implementing this protocol). The MachineId is part of the Hermes configuration.*)
		bFailedBoard : BOOL; (*A value of Unknown Board, Good Board & Failed Board*)
		bProductTypeId : BOOL; (*Identifies a collection of PCBs sharing common properties.*)
		bFlippedBoard : BOOL; (*A value of Unknown Side, Top Side Up & Bottom Side Up.*)
		bTopBarcode : BOOL; (*The barcode of the top side of the next PCB*)
		bBottomBarcode : BOOL; (*The barcode of the bottom side of the next PCB*)
		bLength : BOOL; (*The length of the PCB in millimeter.*)
		bWidth : BOOL; (*The width of the PCB in millimeter.*)
		bThickness : BOOL; (*The thickness of the PCB in millimeter.*)
		bConveyorSpeed : BOOL; (*The conveyor speed preferred by the upstream machine in millimeter per second.*)
		bTopClearanceHeight : BOOL; (*The clearance height for the top side of the PCB in millimeter.*)
		bBottomClearanceHeight : BOOL; (*The clearance height for the bottom side of the PCB in millimeter.*)
		bWeight : BOOL; (*The weight of the PCB in grams.*)
		bWorkOrderId : BOOL; (*The work order for the production of PCB.*)
		bBatchId : BOOL; (*The batch id of a splitted work order.*)
		bRoute : BOOL;
		bAction : BOOL;
	END_STRUCT;
	tyHermesQueryWorkOrderInfoAvl : 	STRUCT
		bQueryId : BOOL; (*Indicates the ID of QueryWorkOrder message. The ID must be unambiguous and e.g. can be a timestamp or a GUID.*)
		bMachineId : BOOL; (*ID / name of this machine for identifying it in a Hermes enabled production line.*)
		bMagazineId : BOOL; (*Barcode of a magazine, required to identify the magazine.*)
		bSlotId : BOOL; (*Indicates the slot in the magazine, enumerated from bottom to top, beginning with 1.*)
		bBarcode : BOOL; (*The barcode of the PCB.*)
	END_STRUCT;
	tyHermesSendWorkOrderInfoAvl : 	STRUCT
		bQueryId : BOOL; (*ID of QueryWorkOrderInfo this message refers to. This attribute is mandatory if it has been in the QueryWorkOrderInfo message.*)
		bWorkOrderId : BOOL; (*Identifies the work order for production of the PCB.*)
		bBatchId : BOOL; (*The batch id of a splitted work order.*)
		bBoardId : BOOL; (*Indicating the ID of the available board.*)
		bBoardIdCreatedBy : BOOL; (*MachineId of the machine which created the BoardId (the first machine in a consecutive row of machines implementing this protocol). The MachineId is part of the Hermes configuration.*)
		bFailedBoard : BOOL; (*A value of Unknown Board, Good Board & Failed Board. This attribute will not be sent if the board information has not been found.*)
		bProductTypeId : BOOL; (*Identifies a collection of PCBs sharing common properties.*)
		bFlippedBoard : BOOL; (*A value of Unknown Side, Top Side Up & Bottom Side Up. This attribute will not be sent if the board information has not been found.*)
		bTopBarcode : BOOL; (*The barcode of the top side of the next PCB. This attribute is mandatory if it has been in the QueryWorkOrderInfo message.*)
		bBottomBarcode : BOOL; (*The barcode of the bottom side of the next PCB. This attribute is mandatory if it has been in the QueryWorkOrderInfo message.*)
		bLength : BOOL; (*The length of the PCB in millimeter.*)
		bWidth : BOOL; (*The width of the PCB in millimeter.*)
		bThickness : BOOL; (*The thickness of the PCB in millimeter.*)
		bConveyorSpeed : BOOL; (*The thickness of the PCB in millimeter.*)
		bTopClearanceHeight : BOOL; (*The clearance height for the top side of the PCB in millimeter.*)
		bBottomClearanceHeight : BOOL; (*The clearance height for the bottom side of the PCB in millimeter.*)
		bWeight : BOOL; (*The weight of the PCB in grams.*)
		bRoute : BOOL;
	END_STRUCT;
	tyHermesCommandAvl : 	STRUCT
		bCommand : BOOL;
	END_STRUCT;
	tyHermesSetConfigurationAvl : 	STRUCT
		bMachineId : BOOL; (*ID/name of this machine for identifying it in a Hermes enabled production line*)
		bSupervisorySystemPort : BOOL; (*Supervisory system port number.*)
		bUpstreamConfigurations : BOOL; (*Upstream configurations*)
		bDownstreamConfigurations : BOOL; (*Downstream configurations*)
		iUpstreamConfigurations : INT; (*Number of upstream configurations*)
		iDownstreamConfigurations : INT; (*Number of downstream configurations*)
		a_tyUpstreamConfigurations : ARRAY[0..c_diHermesConfigMaxIdx]OF tyHermesUpstreamConfigurationAvl; (*Configuration for upstream lanes*)
		a_tyDownstreamConfigurations : ARRAY[0..c_diHermesConfigMaxIdx]OF tyHermesDnstreamConfigurationAvl; (*Configuration for downstream lanes*)
	END_STRUCT;
	tyHermesCurrentConfigurationAvl : 	STRUCT
		bMachineId : BOOL; (*ID/name of this machine for identifying it in a Hermes enabled production line*)
		bSupervisorySystemPort : BOOL; (*Supervisory system port number.*)
		bUpstreamConfigurations : BOOL; (*Upstream configurations*)
		bDownstreamConfigurations : BOOL; (*Downstream configurations*)
		iUpstreamConfigurations : INT; (*Number of upstream configurations*)
		iDownstreamConfigurations : INT; (*Number of downstream configurations*)
		a_tyUpstreamConfigurations : ARRAY[0..c_diHermesConfigMaxIdx]OF tyHermesUpstreamConfigurationAvl; (*Configuration for upstream lanes*)
		a_tyDownstreamConfigurations : ARRAY[0..c_diHermesConfigMaxIdx]OF tyHermesDnstreamConfigurationAvl; (*Configuration for downstream lanes*)
	END_STRUCT;
	tyHermesUpstreamConfigurationAvl : 	STRUCT
		bUpstreamLaneId : BOOL; (*The lane on the upstream side Lanes are enumerated looking downstream from right to left beginning with 1*)
		bUpstreamInterfaceId : BOOL; (*The ID of the transportation interface on the upstream side*)
		bHostAddress : BOOL; (*The IP address or hostname of the upstream machine for this lane and transportation interface*)
		bPort : BOOL; (*Port number on which connections shall be established*)
	END_STRUCT;
	tyHermesDnstreamConfigurationAvl : 	STRUCT
		bDownstreamLaneId : BOOL; (*The lane on the downstream side Lanes are enumerated looking downstream from right to left beginning with 1*)
		bDownstreamInterfaceId : BOOL; (*The ID of the transportation interface on the downstream side*)
		bClientAddress : BOOL; (*The IP address or hostname of the downstream machine for this lane and transportation interface. If not specified, then connections from any IP address are accepted.*)
		bPort : BOOL; (*Port number on which the server shall accept connections for this lane*)
	END_STRUCT;
END_TYPE
```

#### Constants.var - Exported constants
```iecst
VAR CONSTANT
	c_diHermesConfigMaxIdx : DINT := 3; (*Total Config Buffer Size, now is limit at 0~3 = Four*)
	c_diHermesConfigMaxInterfaceIdx : USINT := 2*c_diHermesConfigMaxIdx;
END_VAR
```

#### fbHermesSequenceUS.st
```iecst
(* Hermes Sequence For Upstream *)
FUNCTION_BLOCK fbHermesSequenceUS

	IF (bEn = TRUE) AND (udiStatus >= 65534) THEN

		udiStatus	:= 65535;

		IF (bRstState = TRUE) AND (eState <> HermesStateNotConnected) AND (eState <> HermesStateServiceDescription) THEN
			eState			:= HermesStateNotAvailableNotReady;
			bBoardAvailable	:= FALSE;
		END_IF

		eMsgTypeSnd	:= HermesMsgTypeNA;

		CASE eState OF

			HermesStateNotConnected:
				eMsgTypeSnd	:= HermesMsgTypeServiceDescription;

				eState	:= HermesStateServiceDescription;

			HermesStateServiceDescription:
				IF p_tyMsgTypeRcv.bServiceDescription = TRUE THEN

					p_tyMsgTypeRcv.bServiceDescription	:= FALSE;

					eState	:= HermesStateNotAvailableNotReady;

				END_IF

			HermesStateNotAvailableNotReady:

				IF  bProcessBoardForecastId THEN

					eState	:= HermesStateNotAvailableNotReady;

				ELSIF bRdyRcv = TRUE AND bBlkUS = FALSE THEN //bRdyRcv = Machine in OpsG step USCommTmr (Have USB)

					eMsgTypeSnd	:= HermesMsgTypeMachineReady;

					eState	:= HermesStateMachineReady;

				ELSIF p_tyMsgTypeRcv.bBoardAvailable = TRUE THEN

					p_tyMsgTypeRcv.bBoardAvailable	:= FALSE;

					bBoardAvailable	:= TRUE;

					eState	:= HermesStateBoardAvailable;

				END_IF

			HermesStateBoardAvailable:
				IF bRdyRcv = TRUE AND bBlkUS = FALSE THEN //bRdyRcv = Machine in OpsG step USCommTmr (Have USB)

					eMsgTypeSnd	:= HermesMsgTypeMachineReady;

					eState	:= HermesStateAvailableAndReady;

				ELSIF p_tyMsgTypeRcv.bRevokeBoardAvailable = TRUE THEN

					p_tyMsgTypeRcv.bRevokeBoardAvailable	:= FALSE;

					bBoardAvailable	:= FALSE;

					eState	:= HermesStateNotAvailableNotReady;

				END_IF

			HermesStateMachineReady:

				IF  EDGEPOS(bProcessBoardForecastId) THEN

					eMsgTypeSnd	:= HermesMsgTypeRevokeMachineReady;

					eState	:= HermesStateNotAvailableNotReady;

				ELSIF bRdyRcv = FALSE OR bBlkUS = TRUE THEN //bRdyRcv = Machine in OpsG step USCommTmr (Have USB)

					eMsgTypeSnd	:= HermesMsgTypeRevokeMachineReady;

					eState	:= HermesStateNotAvailableNotReady;

				ELSIF p_tyMsgTypeRcv.bBoardAvailable = TRUE THEN

					p_tyMsgTypeRcv.bBoardAvailable	:= FALSE;

					bBoardAvailable	:= TRUE;

					eState	:= HermesStateAvailableAndReady;

				END_IF

			HermesStateAvailableAndReady:
				IF bRdyRcv = FALSE OR bBlkUS = TRUE THEN

					eMsgTypeSnd	:= HermesMsgTypeRevokeMachineReady;

					eState	:= HermesStateBoardAvailable;

				ELSIF p_tyMsgTypeRcv.bRevokeBoardAvailable = TRUE THEN

					p_tyMsgTypeRcv.bRevokeBoardAvailable	:= FALSE;

					bBoardAvailable	:= FALSE;

					eState	:= HermesStateMachineReady;

				ELSIF bRdyTransport = TRUE AND bBlkUS = FALSE THEN

					eMsgTypeSnd		:= HermesMsgTypeStartTransport;
					bStopTransport	:= FALSE;

					eState	:= HermesStateTransporting;

				END_IF

			HermesStateTransporting:
				IF bRcvCompl OR bRcvIncompl OR bRcvNotStart THEN

					eMsgTypeSnd		:= HermesMsgTypeStopTransport;
					bStopTransport	:= bRcvIncompl OR bRcvNotStart;

					eState	:= HermesStateTransportStopped;

				ELSIF p_tyMsgTypeRcv.bTransportFinished = TRUE THEN

					p_tyMsgTypeRcv.bTransportFinished	:= FALSE;

					eState	:= HermesStateTransportFinished;

				END_IF

				IF p_tyMsgTypeRcv.bBoardAvailable = TRUE THEN

					p_tyMsgTypeRcv.bBoardAvailable	:= FALSE;

					bBoardAvailable	:= TRUE;

				END_IF

				IF p_tyMsgTypeRcv.bRevokeBoardAvailable = TRUE THEN

					p_tyMsgTypeRcv.bRevokeBoardAvailable	:= FALSE;

					bBoardAvailable	:= FALSE;

				END_IF

			HermesStateTransportFinished:
				IF bRcvCompl OR bRcvIncompl OR bRcvNotStart THEN

					eMsgTypeSnd		:= HermesMsgTypeStopTransport;
					bStopTransport	:= bRcvIncompl OR bRcvNotStart;

					eState	:= HermesStateNotAvailableNotReady;

				END_IF

			HermesStateTransportStopped:
				IF p_tyMsgTypeRcv.bTransportFinished = TRUE THEN

					p_tyMsgTypeRcv.bTransportFinished	:= FALSE;

					eState	:= HermesStateNotAvailableNotReady;

				END_IF

				IF p_tyMsgTypeRcv.bBoardAvailable = TRUE THEN

					p_tyMsgTypeRcv.bBoardAvailable	:= FALSE;

					bBoardAvailable	:= TRUE;

				END_IF

				IF p_tyMsgTypeRcv.bRevokeBoardAvailable = TRUE THEN

					p_tyMsgTypeRcv.bRevokeBoardAvailable	:= FALSE;

					bBoardAvailable	:= FALSE;

				END_IF

		END_CASE

		bNotAvlNotRdy   := (eState = HermesStateNotAvailableNotReady);
		bUSRdy			:= (eState = HermesStateBoardAvailable) OR (eState = HermesStateAvailableAndReady) OR (eState >= HermesStateTransporting);
		bDSRdy			:= (eState = HermesStateMachineReady) OR (eState = HermesStateAvailableAndReady) OR (eState >= HermesStateTransporting);
		bTransporting	:= eState >= HermesStateTransporting;

	ELSIF (bEn = FALSE) AND (udiStatus <> 65534) THEN

		udiStatus	:= 65534;

		bBoardAvailable	:= FALSE;
		bUSRdy			:= FALSE;
		bDSRdy			:= FALSE;
		bTransporting	:= FALSE;
		bStopTransport	:= FALSE;
		eState			:= HermesStateNotConnected;

	END_IF

END_FUNCTION_BLOCK
```

#### fbHermesSequenceDS.st
```iecst
(* Hermes Sequence For Downstream *)
FUNCTION_BLOCK fbHermesSequenceDS

	IF (bEn = TRUE) AND (udiStatus >= 65534) THEN

		udiStatus	:= 65535;

		IF (bRstState = TRUE) AND (eState <> HermesStateNotConnected) AND (eState <> HermesStateServiceDescription) THEN
			eState	:= HermesStateNotAvailableNotReady;
		END_IF

		eMsgTypeSnd	:= HermesMsgTypeNA;

		CASE eState OF

			HermesStateNotConnected:
				IF p_tyMsgTypeRcv.bServiceDescription = TRUE THEN

					p_tyMsgTypeRcv.bServiceDescription	:= FALSE;

					eState	:= HermesStateServiceDescription;

				END_IF

			HermesStateServiceDescription:
				eMsgTypeSnd	:= HermesMsgTypeServiceDescription;

				eState	:= HermesStateNotAvailableNotReady;

			HermesStateNotAvailableNotReady:

				IF bFeatureBoardForecast = TRUE THEN
					IF bOpsRun THEN
						IF  bSendBFId = TRUE AND bBFIdSent = FALSE THEN
							eMsgTypeSnd	:= HermesMsgTypeBoardForecastId; //Send BoardForecast(Id) after a Changeover with all zones free

						ELSIF bSendBFId = FALSE  AND EDGEPOS(bSendBFNoID) THEN
							eMsgTypeSnd	:= HermesMsgTypeBoardForecastNoId; //Send BoardForecast() when PCB_In (Have Board) at first zone

						END_IF
					END_IF
				END_IF

				IF bRdySnd = TRUE AND bBlkDS = FALSE AND bSendBFId = FALSE (*AND bFirstZoneEndSen*) AND bFeatureBoardForecast = TRUE THEN

					eMsgTypeSnd	:= HermesMsgTypeBoardAvailable;

					eState	:= HermesStateBoardAvailable;

				ELSIF bRdySnd = TRUE AND bBlkDS  = FALSE AND bSendBFId = FALSE AND bFeatureBoardForecast = FALSE  THEN

						eMsgTypeSnd	:= HermesMsgTypeBoardAvailable;

						eState	:= HermesStateBoardAvailable;

				ELSIF p_tyMsgTypeRcv.bMachineReady = TRUE THEN

					p_tyMsgTypeRcv.bMachineReady	:= FALSE;

					eState	:= HermesStateMachineReady;

				END_IF

			HermesStateBoardAvailable:
				IF (bRdySnd = FALSE OR bBlkDS = TRUE) AND bSendBFId = FALSE THEN

					eMsgTypeSnd	:= HermesMsgTypeRevokeBoardAvl;

					eState	:= HermesStateNotAvailableNotReady;

				ELSIF p_tyMsgTypeRcv.bMachineReady = TRUE THEN

					p_tyMsgTypeRcv.bMachineReady	:= FALSE;

					eState	:= HermesStateAvailableAndReady;

				END_IF

			HermesStateMachineReady:

				IF bFeatureBoardForecast = TRUE THEN
					IF bOpsRun THEN
						IF bSendBFId = TRUE AND bBFIdSent = FALSE  THEN
							eMsgTypeSnd	:= HermesMsgTypeBoardForecastId; //Send BoardForecast(Id) after a Changeover with all zones free

						ELSIF  bSendBFId = FALSE  AND EDGEPOS(bSendBFNoID) THEN

							eMsgTypeSnd	:= HermesMsgTypeBoardForecastNoId; //Send BoardForecast() when PCB_In (Have Board) at first zone

						END_IF
					END_IF

				END_IF

				IF (bRdySnd = TRUE AND bBlkDS = FALSE )AND bSendBFId = FALSE (*AND bFirstZoneEndSen*) AND bFeatureBoardForecast = TRUE THEN

					eMsgTypeSnd	:= HermesMsgTypeBoardAvailable;

					eState	:= HermesStateAvailableAndReady;

				ELSIF (bRdySnd = TRUE AND bBlkDS = FALSE ) AND bSendBFId = FALSE AND bFeatureBoardForecast = FALSE  THEN

					eMsgTypeSnd	:= HermesMsgTypeBoardAvailable;

					eState	:= HermesStateAvailableAndReady;

				ELSIF p_tyMsgTypeRcv.bRevokeMachineReady = TRUE THEN

					p_tyMsgTypeRcv.bRevokeMachineReady	:= FALSE;

					eState	:= HermesStateNotAvailableNotReady;

				ELSIF p_tyMsgTypeRcv.bStartTransport = TRUE AND bSendBFId = FALSE THEN

					p_tyMsgTypeRcv.bStartTransport	:= FALSE;
					bStopTransport					:= FALSE;

					eState	:= HermesStateTransporting;

				END_IF

			HermesStateAvailableAndReady:
				IF bRdySnd = FALSE  OR  bBlkDS = TRUE THEN

					eMsgTypeSnd	:= HermesMsgTypeRevokeBoardAvl;

					eState	:= HermesStateMachineReady;

				ELSIF p_tyMsgTypeRcv.bRevokeMachineReady = TRUE THEN

					p_tyMsgTypeRcv.bRevokeMachineReady	:= FALSE;

					eState	:= HermesStateBoardAvailable;

				ELSIF p_tyMsgTypeRcv.bStartTransport = TRUE THEN

					p_tyMsgTypeRcv.bStartTransport	:= FALSE;
					bStopTransport					:= FALSE;

					eState	:= HermesStateTransporting;

				END_IF

			HermesStateTransporting:
				IF bSndCompl OR bSndIncompl OR bSndNotStart THEN

					eMsgTypeSnd		:= HermesMsgTypeTransportFinished;
					bStopTransport	:= bSndIncompl OR bSndNotStart;

					eState	:= HermesStateTransportFinished;

				ELSIF p_tyMsgTypeRcv.bStopTransport = TRUE THEN

					p_tyMsgTypeRcv.bStopTransport	:= FALSE;

					eState	:= HermesStateTransportStopped;

				END_IF

			HermesStateTransportFinished:
				IF p_tyMsgTypeRcv.bStopTransport = TRUE THEN

					p_tyMsgTypeRcv.bStopTransport	:= FALSE;

					eState	:= HermesStateNotAvailableNotReady;

				END_IF

			HermesStateTransportStopped:
				IF bSndCompl OR bSndIncompl OR bSndNotStart THEN

					eMsgTypeSnd		:= HermesMsgTypeTransportFinished;
					bStopTransport	:= bSndIncompl OR bSndNotStart;

					eState	:= HermesStateNotAvailableNotReady;

				END_IF

		END_CASE

		bUSRdy			:= (eState = HermesStateBoardAvailable) OR (eState = HermesStateAvailableAndReady) OR (eState >= HermesStateTransporting);
		bDSRdy			:= (eState = HermesStateMachineReady) OR (eState = HermesStateAvailableAndReady) OR (eState >= HermesStateTransporting);
		bTransporting	:= eState >= HermesStateTransporting;

	ELSIF (bEn = FALSE) AND (udiStatus <> 65534) THEN

		udiStatus	:= 65534;

		bUSRdy			:= FALSE;
		bDSRdy			:= FALSE;
		bTransporting	:= FALSE;
		bStopTransport	:= FALSE;

		eState	:= HermesStateNotConnected;

	END_IF

END_FUNCTION_BLOCK
```

#### fbHermesSequenceSvy.st
```iecst
(* Hermes Sequence For Supervisory System *)
FUNCTION_BLOCK fbHermesSequenceSvy

	IF (bEn = TRUE) AND (udiStatus >= 65534) THEN

		udiStatus	:= 65535;

		IF (bRstState = TRUE) AND (eState <> HermesStateNotConnected) AND (eState <> HermesStateSServiceDescription) THEN
			eState	:= HermesStateConnected;
		END_IF

		eMsgTypeSnd	:= HermesMsgTypeNA;

		CASE eState OF

			HermesStateNotConnected:
				IF p_tyMsgTypeRcv.bSServiceDescription = TRUE THEN

					p_tyMsgTypeRcv.bSServiceDescription	:= FALSE;

					eState	:= HermesStateSServiceDescription;

				END_IF

			HermesStateSServiceDescription:
				eMsgTypeSnd	:= HermesMsgTypeSServiceDescription;

				eState	:= HermesStateConnected;

			HermesStateConnected:
				IF p_tyMsgTypeRcv.bGetConfiguration = TRUE THEN

					p_tyMsgTypeRcv.bGetConfiguration	:= FALSE;

					eMsgTypeSnd	:= HermesMsgTypeCurrConfiguration;

				END_IF

		END_CASE

	ELSIF (bEn = FALSE) AND (udiStatus <> 65534) THEN

		udiStatus	:= 65534;

		eState	:= HermesStateNotConnected;

	END_IF

END_FUNCTION_BLOCK
```

#### fbHermesSequenceTO.st
```iecst
(* Hermes Sequence Time Out *)
FUNCTION_BLOCK fbHermesSequenceTO

	IF (bEn = TRUE) AND (udiStatus >= 65534) THEN

		udiStatus	:= 65535;

		IF (eState = HermesStateNotConnected) OR (eState = HermesStateServiceDescription) THEN
			fbConnTimeOut(IN := TRUE , PT := tConnTimeOut);
		END_IF

		IF (eState = HermesStateTransporting) OR (eState = HermesStateTransportFinished) OR (eState = HermesStateTransportStopped) THEN
			fbTransportTimeOut(IN := TRUE , PT := tTransportTimeOut);
		END_IF

		IF eState = HermesStateNotAvailableNotReady THEN
			fbConnTimeOut(IN := FALSE);
			fbTransportTimeOut(IN := FALSE);
		END_IF

		IF fbConnTimeOut.Q = TRUE THEN
			udiStatus	:= 2912;	//Connection Time Out
		ELSIF fbTransportTimeOut.Q = TRUE THEN
			udiStatus	:= 2913;	//Transport Time Out
		END_IF

	ELSIF (bEn = FALSE) AND (udiStatus <> 65534) THEN

		udiStatus	:= 65534;

		fbConnTimeOut(IN := FALSE);
		fbTransportTimeOut(IN := FALSE);
	END_IF

END_FUNCTION_BLOCK
```

#### fbHermesSequenceSvyTO.st
```iecst
(* Hermes Sequence Supervisory Time Out *)
FUNCTION_BLOCK fbHermesSequenceSvyTO

	IF (bEn = TRUE) AND (udiStatus >= 65534) THEN

		udiStatus	:= 65535;

		IF (eState = HermesStateNotConnected) OR (eState = HermesStateSServiceDescription) THEN
			fbConnTimeOut(IN := TRUE , PT := tConnTimeOut);
		END_IF

		IF  eState = HermesStateConnected THEN
			fbConnTimeOut(IN := FALSE);
		END_IF

		IF fbConnTimeOut.Q = TRUE THEN
			udiStatus	:= 2912;	//Connection Time Out
		END_IF

	ELSIF (bEn = FALSE) AND (udiStatus <> 65534) THEN

		udiStatus	:= 65534;

		fbConnTimeOut(IN := FALSE);
	END_IF

END_FUNCTION_BLOCK
```

#### fHermesCmpSlt.st
```iecst
(* Hermes Compare Slot Parameter *)
FUNCTION fHermesCmpSlt

	fHermesCmpSlt	:= 0;

	IF diRcpMinSltValue <= 0 THEN
		fHermesCmpSlt	:= 2914;	//Input First Slot Is Invalid

	ELSIF diRcpMaxSltValue <= 0 THEN
		fHermesCmpSlt	:= 2915;	//Input Last Slot Is Invalid

	ELSIF diRcpPitch <= 0 THEN
		fHermesCmpSlt	:= 2916;	//Input Pitch Is Invalid

	ELSIF diRcpSltToSltInUM <= 0 THEN
		fHermesCmpSlt	:= 2917;	//Input Slot To Slot Distance Is Invalid

	ELSIF diRcpTtlSlt <= 0 THEN
		fHermesCmpSlt	:= 2918;	//Input Total Slot Is Invalid

	ELSIF rHermesThicknessInMM <= 0 THEN
		fHermesCmpSlt	:= 2919;	//Input Thickness Is Invalid

	ELSIF rHermesTopClearanceHeightInMM <= 0 THEN
		fHermesCmpSlt	:= 2920;	//Input Top Clearance Height Is Invalid

	ELSIF rHermesBtmClearanceHeightInMM <= 0 THEN
		fHermesCmpSlt	:= 2921;	//Input Bottom Clearance Height Is Invalid

	ELSE
		fbGetSlt.eFlippedBrd				:= eHermesFlippedBrd;
		fbGetSlt.rThicknessInMM				:= rHermesThicknessInMM;
		fbGetSlt.rTopClearanceHeightInMM	:= rHermesTopClearanceHeightInMM;
		fbGetSlt.rBtmClearanceHeightInMM	:= rHermesBtmClearanceHeightInMM;
		fbGetSlt.diSltToSltInUM				:= diRcpSltToSltInUM;
		fbGetSlt.diTtlSlt					:= diRcpTtlSlt;
		fbGetSlt;

		IF (fHermesCmpSlt = 0) THEN
			IF diRcpMinSltValue < fbGetSlt.diMinSltValue THEN
				fHermesCmpSlt	:= 2922;	//Recipe First Slot Value & Board Available Data Not Match
			END_IF
		END_IF

		IF (fHermesCmpSlt = 0) THEN
			IF diRcpMaxSltValue > fbGetSlt.diMaxSltValue THEN
				fHermesCmpSlt	:= 2923;	//Recipe Last Slot Value & Board Available Data Not Match
			END_IF
		END_IF

		IF (fHermesCmpSlt = 0) THEN
			IF diRcpPitch < fbGetSlt.diPitch THEN
				fHermesCmpSlt	:= 2924;	//Recipe Pitch Value & Board Available Data Not Match
			END_IF
		END_IF

	END_IF

END_FUNCTION
```

#### fbHermesGetSlt.st
```iecst
(* Hermes Get Slot Parameter *)
FUNCTION_BLOCK fbHermesGetSlt

	IF (rThicknessInMM <= 0) OR (rTopClearanceHeightInMM <= 0) OR (rBtmClearanceHeightInMM <= 0) OR (diTtlSlt <= 0) OR (diSltToSltInUM <= 0) THEN
		diMinSltValue	:= 0;
		diMaxSltValue	:= 0;
		diPitch			:= 0;
		diSltToSltInUM	:= 0;

	ELSE
		diThicknessInUM				:= REAL_TO_DINT(rThicknessInMM * 1000);
		diTopClearanceHeightInUM	:= REAL_TO_DINT(rTopClearanceHeightInMM * 1000);
		diBtmClearanceHeightInUM	:= REAL_TO_DINT(rBtmClearanceHeightInMM * 1000);

		IF eFlippedBrd = HermesFlippedBoardBtmSideUp THEN

			diMinSltValue	:= (diTopClearanceHeightInUM / diSltToSltInUM) + 1;
			diMaxSltValue	:= diTtlSlt - ((diBtmClearanceHeightInUM + diThicknessInUM) / diSltToSltInUM);
			diPitch			:= ((diTopClearanceHeightInUM + diBtmClearanceHeightInUM + diThicknessInUM) / diSltToSltInUM) + 1;

		ELSE

			diMinSltValue	:= (diBtmClearanceHeightInUM / diSltToSltInUM) + 1;
			diMaxSltValue	:= diTtlSlt - ((diTopClearanceHeightInUM + diThicknessInUM) / diSltToSltInUM);
			diPitch			:= ((diTopClearanceHeightInUM + diBtmClearanceHeightInUM + diThicknessInUM) / diSltToSltInUM) + 1;

		END_IF

	END_IF

END_FUNCTION_BLOCK
```

#### fbHermesGetSndConfig.st
```iecst
(* Hermes Get & Send Configuration *)
FUNCTION_BLOCK fbHermesGetSndConfig

	IF (bEn = TRUE) AND (udiStatus >= 65534) THEN

		udiStatus	:= 65535;

		IF p_tyMsgTypeRcv.bGetConfiguration = TRUE THEN

			p_tyMsgTypeRcv.bGetConfiguration	:= FALSE;

			p_tyMsgTypeSnd.bCurrentConfiguration	:= TRUE;

			tyCurrentConfiguration.tyData	:= tyCurrentConfigurationData;

			IF tyCurrentConfiguration.tyData.sMachineId <> '' THEN
				tyCurrentConfiguration.tyAvl.bMachineId	:= TRUE;
			END_IF

			FOR di := 0 TO c_diHermesConfigMaxIdx DO

				IF tyCurrentConfiguration.tyData.a_tyUpstreamConfigurations[di].iUpstreamLaneId <> 0 THEN
					tyCurrentConfiguration.tyAvl.a_tyUpstreamConfigurations[di].bUpstreamLaneId	:= TRUE;
					tyCurrentConfiguration.tyAvl.bUpstreamConfigurations	:= TRUE;
					tyCurrentConfiguration.tyAvl.iUpstreamConfigurations	:= DINT_TO_INT(di) + 1;

					IF tyCurrentConfiguration.tyData.a_tyUpstreamConfigurations[di].sUpstreamInterfaceId <> '' THEN
						tyCurrentConfiguration.tyAvl.a_tyUpstreamConfigurations[di].bUpstreamInterfaceId	:= TRUE;
					END_IF

					IF tyCurrentConfiguration.tyData.a_tyUpstreamConfigurations[di].sHostAddress <> '' THEN
						tyCurrentConfiguration.tyAvl.a_tyUpstreamConfigurations[di].bHostAddress	:= TRUE;
					END_IF

					IF tyCurrentConfiguration.tyData.a_tyUpstreamConfigurations[di].uiPort <> 0 THEN
						tyCurrentConfiguration.tyAvl.a_tyUpstreamConfigurations[di].bPort	:= TRUE;
					END_IF

				ELSE

					EXIT;

				END_IF

			END_FOR

			FOR di := 0 TO c_diHermesConfigMaxIdx DO

				IF tyCurrentConfiguration.tyData.a_tyDownstreamConfigurations[di].iDownstreamLaneId <> 0 THEN
					tyCurrentConfiguration.tyAvl.a_tyDownstreamConfigurations[di].bDownstreamLaneId	:= TRUE;
					tyCurrentConfiguration.tyAvl.bDownstreamConfigurations	:= TRUE;
					tyCurrentConfiguration.tyAvl.iDownstreamConfigurations	:= DINT_TO_INT(di) + 1;

					IF tyCurrentConfiguration.tyData.a_tyDownstreamConfigurations[di].sDownstreamInterfaceId <> '' THEN
						tyCurrentConfiguration.tyAvl.a_tyDownstreamConfigurations[di].bDownstreamInterfaceId	:= TRUE;
					END_IF

					IF tyCurrentConfiguration.tyData.a_tyDownstreamConfigurations[di].sClientAddress <> '' THEN
						tyCurrentConfiguration.tyAvl.a_tyDownstreamConfigurations[di].bClientAddress	:= TRUE;
					END_IF

					IF tyCurrentConfiguration.tyData.a_tyDownstreamConfigurations[di].uiPort <> 0 THEN
						tyCurrentConfiguration.tyAvl.a_tyDownstreamConfigurations[di].bPort	:= TRUE;
					END_IF

				ELSE

					EXIT;

				END_IF

			END_FOR

		END_IF

	ELSIF (bEn = FALSE) AND (udiStatus <> 65534) THEN

		udiStatus	:= 65534;

		memset(ADR(tyCurrentConfiguration) , 0 , SIZEOF(tyCurrentConfiguration));

	END_IF

END_FUNCTION_BLOCK
```

#### fbHermesParseXMLTable.st
```iecst
(* Hermes Parse XML Table Data *)
FUNCTION_BLOCK fbHermesParseXMLTable

	memset(ADR(tyMsgType) , 0 , SIZEOF(tyMsgType));
	memset(ADR(tyCheckAlive) , 0 , SIZEOF(tyCheckAlive));
	memset(ADR(tyCheckAlivePing) , 0 , SIZEOF(tyCheckAlivePing));
	memset(ADR(tyCheckAlivePong) , 0 , SIZEOF(tyCheckAlivePong));
	memset(ADR(tyServiceDescription) , 0 , SIZEOF(tyServiceDescription));
	memset(ADR(tySServiceDescription) , 0 , SIZEOF(tySServiceDescription));
	memset(ADR(tyNotification) , 0 , SIZEOF(tyNotification));
	memset(ADR(tyBoardAvailable) , 0 , SIZEOF(tyBoardAvailable));
	memset(ADR(tyMachineReady) , 0 , SIZEOF(tyMachineReady));
	memset(ADR(tyStartTransport) , 0 , SIZEOF(tyStartTransport));
	memset(ADR(tyStopTransport) , 0 , SIZEOF(tyStopTransport));
	memset(ADR(tyTransportFinished) , 0 , SIZEOF(tyTransportFinished));
	memset(ADR(tySetConfiguration) , 0 , SIZEOF(tySetConfiguration));
	memset(ADR(tyCurrentConfiguration) , 0 , SIZEOF(tyCurrentConfiguration));
	memset(ADR(tyBoardForecast) , 0 , SIZEOF(tyBoardForecast));
	memset(ADR(tyBoardArrived) , 0 , SIZEOF(tyBoardArrived));
	memset(ADR(tyBoardDeparted) , 0 , SIZEOF(tyBoardDeparted));
	memset(ADR(tyQueryBoardInfo) , 0 , SIZEOF(tyQueryBoardInfo));
	memset(ADR(tySendBoardInfo) , 0 , SIZEOF(tySendBoardInfo));
	memset(ADR(tyQueryWorkOrderInfo) , 0 , SIZEOF(tyQueryWorkOrderInfo));
	memset(ADR(tySendWorkOrderInfo) , 0 , SIZEOF(tySendWorkOrderInfo));
	memset(ADR(tyCommand),0,SIZEOF(tyCommand));

	iCheckAliveFirstIdx				:= -1;
	iCheckAliveLastIdx				:= -1;
	iCheckAlivePingFirstIdx			:= -1;
	iCheckAlivePingLastIdx			:= -1;
	iCheckAlivePongFirstIdx			:= -1;
	iCheckAlivePongLastIdx			:= -1;
	iServiceDescriptionFirstIdx		:= -1;
	iServiceDescriptionLastIdx		:= -1;
	iSServiceDescriptionFirstIdx	:= -1;
	iSServiceDescriptionLastIdx  	:= -1;
	iNotificationFirstIdx			:= -1;
	iNotificationLastIdx			:= -1;
	iBoardAvailableFirstIdx			:= -1;
	iBoardAvailableLastIdx			:= -1;
	iRevokeBoardAvailableFirstIdx	:= -1;
	iRevokeBoardAvailableLastIdx	:= -1;
	iMachineReadyFirstIdx			:= -1;
	iMachineReadyLastIdx			:= -1;
	iRevokeMachineReadyFirstIdx		:= -1;
	iRevokeMachineReadyLastIdx		:= -1;
	iStartTransportFirstIdx			:= -1;
	iStartTransportLastIdx			:= -1;
	iStopTransportFirstIdx			:= -1;
	iStopTransportLastIdx			:= -1;
	iTransportFinishedFirstIdx		:= -1;
	iTransportFinishedLastIdx		:= -1;
	iSetConfigurationFirstIdx		:= -1;
	iSetConfigurationLastIdx		:= -1;
	iGetConfigurationFirstIdx		:= -1;
	iGetConfigurationLastIdx		:= -1;
	iCurrentConfigurationFirstIdx	:= -1;
	iCurrentConfigurationLastIdx	:= -1;
	iBoardForecastFirstIdx			:= -1;
	iBoardForecastLastIdx			:= -1;
	iBoardArrivedFirstIdx			:= -1;
	iBoardArrivedLastIdx			:= -1;
	iBoardDepartedFirstIdx			:= -1;
	iBoardDepartedLastIdx			:= -1;
	iQueryBoardInfoFirstIdx			:= -1;
	iQueryBoardInfoLastIdx			:= -1;
	iSendBoardInfoFirstIdx			:= -1;
	iSendBoardInfoLastIdx			:= -1;
	iQueryWorkOrderInfoFirstIdx		:= -1;
	iQueryWorkOrderInfoLastIdx		:= -1;
	iSendWorkOrderInfoFirstIdx		:= -1;
	iSendWorkOrderInfoLastIdx		:= -1;
	iCommandFirstIdx				:= -1;
	iCommandLastIdx1				:= -1;
	iHermesIdx						:= -1;

	//iSubBoardCntr
	iSubBoardCntr				    := -1;

	eMsgType	:= HermesMsgTypeNA;

	FOR udi := p_XMLTable TO (p_XMLTable + ((iTotalIdxWrite - 2) * SIZEOF(p_tyXMLTable))) BY SIZEOF(p_tyXMLTable) DO

		p_tyXMLTable ACCESS udi;
		p_tyXMLTable1 ACCESS (udi + SIZEOF(p_tyXMLTable));

		fConvertToLower_254(ADR(sLowerCase) , p_tyXMLTable.sValue);

		IF (p_tyXMLTable.sTitle = 'ST') AND (sLowerCase = 'hermes') THEN

			eMsgType	:= HermesMsgTypeNA;
			iHermesIdx	:= UDINT_TO_INT((udi - p_XMLTable) / (SIZEOF(p_tyXMLTable)));

		ELSIF (p_tyXMLTable.sTitle = 'ET') AND (sLowerCase = 'hermes') THEN

			iHermesIdx	:= -1;

			CASE eMsgType OF

				HermesMsgTypeCheckAlive:
					iCheckAliveLastIdx	:= UDINT_TO_INT(((udi - p_XMLTable) / (SIZEOF(p_tyXMLTable))) + 1);

					IF tyCheckAlive.tyAvl.bType = TRUE AND tyCheckAlive.tyData.eType = HermesCheckAliveTypePing THEN
						tyMsgType.bCheckAlivePing	:= TRUE;
						tyCheckAlivePing			:= tyCheckAlive;
						iCheckAlivePingFirstIdx		:= iCheckAliveFirstIdx;
						iCheckAlivePingLastIdx		:= iCheckAliveLastIdx;

						memset(ADR(tyCheckAlive) , 0 , SIZEOF(tyCheckAlive));
						tyMsgType.bCheckAlive	:= FALSE;
						iCheckAliveFirstIdx		:= -1;
						iCheckAliveLastIdx		:= -1;

					ELSIF tyCheckAlive.tyAvl.bType = TRUE AND tyCheckAlive.tyData.eType = HermesCheckAliveTypePong THEN
						tyMsgType.bCheckAlivePong	:= TRUE;
						tyCheckAlivePong			:= tyCheckAlive;
						iCheckAlivePongFirstIdx		:= iCheckAliveFirstIdx;
						iCheckAlivePongLastIdx		:= iCheckAliveLastIdx;

						memset(ADR(tyCheckAlive) , 0 , SIZEOF(tyCheckAlive));
						tyMsgType.bCheckAlive	:= FALSE;
						iCheckAliveFirstIdx		:= -1;
						iCheckAliveLastIdx		:= -1;

					END_IF

				HermesMsgTypeServiceDescription:	iServiceDescriptionLastIdx		:= UDINT_TO_INT(((udi - p_XMLTable) / (SIZEOF(p_tyXMLTable))) + 1);
				HermesMsgTypeSServiceDescription:	iSServiceDescriptionLastIdx	    := UDINT_TO_INT(((udi - p_XMLTable) / (SIZEOF(p_tyXMLTable))) + 1);
				HermesMsgTypeNotification:			iNotificationLastIdx			:= UDINT_TO_INT(((udi - p_XMLTable) / (SIZEOF(p_tyXMLTable))) + 1);
				HermesMsgTypeBoardAvailable:		iBoardAvailableLastIdx			:= UDINT_TO_INT(((udi - p_XMLTable) / (SIZEOF(p_tyXMLTable))) + 1);
				HermesMsgTypeRevokeBoardAvl:		iRevokeBoardAvailableLastIdx	:= UDINT_TO_INT(((udi - p_XMLTable) / (SIZEOF(p_tyXMLTable))) + 1);
				HermesMsgTypeMachineReady:			iMachineReadyLastIdx			:= UDINT_TO_INT(((udi - p_XMLTable) / (SIZEOF(p_tyXMLTable))) + 1);
				HermesMsgTypeRevokeMachineReady:	iRevokeMachineReadyLastIdx		:= UDINT_TO_INT(((udi - p_XMLTable) / (SIZEOF(p_tyXMLTable))) + 1);
				HermesMsgTypeStartTransport:		iStartTransportLastIdx			:= UDINT_TO_INT(((udi - p_XMLTable) / (SIZEOF(p_tyXMLTable))) + 1);
				HermesMsgTypeStopTransport:			iStopTransportLastIdx			:= UDINT_TO_INT(((udi - p_XMLTable) / (SIZEOF(p_tyXMLTable))) + 1);
				HermesMsgTypeTransportFinished:		iTransportFinishedLastIdx		:= UDINT_TO_INT(((udi - p_XMLTable) / (SIZEOF(p_tyXMLTable))) + 1);
				HermesMsgTypeSetConfiguration:		iSetConfigurationLastIdx		:= UDINT_TO_INT(((udi - p_XMLTable) / (SIZEOF(p_tyXMLTable))) + 1);
				HermesMsgTypeGetConfiguration:		iGetConfigurationLastIdx		:= UDINT_TO_INT(((udi - p_XMLTable) / (SIZEOF(p_tyXMLTable))) + 1);
				HermesMsgTypeCurrConfiguration:		iCurrentConfigurationLastIdx	:= UDINT_TO_INT(((udi - p_XMLTable) / (SIZEOF(p_tyXMLTable))) + 1);
				HermesMsgTypeBoardForecast:			iBoardForecastLastIdx			:= UDINT_TO_INT(((udi - p_XMLTable) / (SIZEOF(p_tyXMLTable))) + 1);
				HermesMsgTypeBoardArrived:			iBoardArrivedLastIdx			:= UDINT_TO_INT(((udi - p_XMLTable) / (SIZEOF(p_tyXMLTable))) + 1);
				HermesMsgTypeBoardDeparted:			iBoardDepartedLastIdx			:= UDINT_TO_INT(((udi - p_XMLTable) / (SIZEOF(p_tyXMLTable))) + 1);
				HermesMsgTypeQueryBoardInfo:		iQueryBoardInfoLastIdx			:= UDINT_TO_INT(((udi - p_XMLTable) / (SIZEOF(p_tyXMLTable))) + 1);
				HermesMsgTypeSendBoardInfo:			iSendBoardInfoLastIdx			:= UDINT_TO_INT(((udi - p_XMLTable) / (SIZEOF(p_tyXMLTable))) + 1);
				HermesMsgTypeQueryWorkOrderInfo:	iQueryWorkOrderInfoLastIdx		:= UDINT_TO_INT(((udi - p_XMLTable) / (SIZEOF(p_tyXMLTable))) + 1);
				HermesMsgTypeSendWorkOrderInfo:		iSendWorkOrderInfoLastIdx		:= UDINT_TO_INT(((udi - p_XMLTable) / (SIZEOF(p_tyXMLTable))) + 1);

			END_CASE

			eMsgType	:= HermesMsgTypeNA;

		ELSIF (p_tyXMLTable.sTitle = 'ST') AND (sLowerCase = 'checkalive') THEN

			eMsgType				:= HermesMsgTypeCheckAlive;
			tyMsgType.bCheckAlive	:= TRUE;
			iCheckAliveFirstIdx		:= iHermesIdx;

		ELSIF (p_tyXMLTable.sTitle = 'ST') AND (sLowerCase = 'servicedescription') THEN

			eMsgType						    := HermesMsgTypeServiceDescription;
			tyMsgType.bServiceDescription    	:= TRUE;
			iServiceDescriptionFirstIdx	     	:= iHermesIdx;

		ELSIF (p_tyXMLTable.sTitle = 'ST') AND (sLowerCase = 'supervisoryservicedescription') THEN

			eMsgType					    	:= HermesMsgTypeSServiceDescription;
			tyMsgType.bSServiceDescription   	:= TRUE;
			iSServiceDescriptionFirstIdx	    := iHermesIdx;

		ELSIF (p_tyXMLTable.sTitle = 'ST') AND (sLowerCase = 'notification') THEN

			eMsgType				:= HermesMsgTypeNotification;
			tyMsgType.bNotification	:= TRUE;
			iNotificationFirstIdx	:= iHermesIdx;

		ELSIF (p_tyXMLTable.sTitle = 'ST') AND (sLowerCase = 'boardavailable') THEN

			eMsgType					:= HermesMsgTypeBoardAvailable;
			tyMsgType.bBoardAvailable	:= TRUE;
			iBoardAvailableFirstIdx		:= iHermesIdx;

		ELSIF (p_tyXMLTable.sTitle = 'ST') AND (sLowerCase = 'revokeboardavailable') THEN

			eMsgType						:= HermesMsgTypeRevokeBoardAvl;
			tyMsgType.bRevokeBoardAvailable	:= TRUE;
			iRevokeBoardAvailableFirstIdx	:= iHermesIdx;

		ELSIF (p_tyXMLTable.sTitle = 'ST') AND (sLowerCase = 'machineready') THEN

			eMsgType				:= HermesMsgTypeMachineReady;
			tyMsgType.bMachineReady	:= TRUE;
			iMachineReadyFirstIdx	:= iHermesIdx;

		ELSIF (p_tyXMLTable.sTitle = 'ST') AND (sLowerCase = 'revokemachineready') THEN

			eMsgType						:= HermesMsgTypeRevokeMachineReady;
			tyMsgType.bRevokeMachineReady	:= TRUE;
			iRevokeMachineReadyFirstIdx		:= iHermesIdx;

		ELSIF (p_tyXMLTable.sTitle = 'ST') AND (sLowerCase = 'starttransport') THEN

			eMsgType					:= HermesMsgTypeStartTransport;
			tyMsgType.bStartTransport	:= TRUE;
			iStartTransportFirstIdx		:= iHermesIdx;

		ELSIF (p_tyXMLTable.sTitle = 'ST') AND (sLowerCase = 'stoptransport') THEN

			eMsgType					:= HermesMsgTypeStopTransport;
			tyMsgType.bStopTransport	:= TRUE;
			iStopTransportFirstIdx		:= iHermesIdx;

		ELSIF (p_tyXMLTable.sTitle = 'ST') AND (sLowerCase = 'transportfinished') THEN

			eMsgType						:= HermesMsgTypeTransportFinished;
			tyMsgType.bTransportFinished	:= TRUE;
			iTransportFinishedFirstIdx		:= iHermesIdx;

		ELSIF (p_tyXMLTable.sTitle = 'ST') AND (sLowerCase = 'setconfiguration') THEN

			eMsgType					:= HermesMsgTypeSetConfiguration;
			tyMsgType.bSetConfiguration	:= TRUE;
			iSetConfigurationFirstIdx	:= iHermesIdx;
			bSetUpstream				:= FALSE;
			bSetDownstream				:= FALSE;

		ELSIF (p_tyXMLTable.sTitle = 'ST') AND (sLowerCase = 'getconfiguration') THEN

			eMsgType					:= HermesMsgTypeGetConfiguration;
			tyMsgType.bGetConfiguration	:= TRUE;
			iGetConfigurationFirstIdx	:= iHermesIdx;

		ELSIF (p_tyXMLTable.sTitle = 'ST') AND (sLowerCase = 'currentconfiguration') THEN

			eMsgType						:= HermesMsgTypeCurrConfiguration;
			tyMsgType.bCurrentConfiguration	:= TRUE;
			iCurrentConfigurationFirstIdx	:= iHermesIdx;
			bCurrUpstream					:= FALSE;
			bCurrDownstream					:= FALSE;

		ELSIF (p_tyXMLTable.sTitle = 'ST') AND (sLowerCase = 'boardforecast') THEN

			eMsgType					:= HermesMsgTypeBoardForecast;
			tyMsgType.bBoardForecast	:= TRUE;
			iBoardForecastFirstIdx		:= iHermesIdx;

		ELSIF (p_tyXMLTable.sTitle = 'ST') AND (sLowerCase = 'boardarrived') THEN

			eMsgType					:= HermesMsgTypeBoardArrived;
			tyMsgType.bBoardArrived	:= TRUE;
			iBoardArrivedFirstIdx		:= iHermesIdx;

		ELSIF (p_tyXMLTable.sTitle = 'ST') AND (sLowerCase = 'boarddeparted') THEN

			eMsgType					:= HermesMsgTypeBoardDeparted;
			tyMsgType.bBoardDeparted	:= TRUE;
			iBoardDepartedFirstIdx		:= iHermesIdx;

		ELSIF (p_tyXMLTable.sTitle = 'ST') AND (sLowerCase = 'queryboardinfo') THEN

			eMsgType					:= HermesMsgTypeQueryBoardInfo;
			tyMsgType.bQueryBoardInfo	:= TRUE;
			iQueryBoardInfoFirstIdx		:= iHermesIdx;

		ELSIF (p_tyXMLTable.sTitle = 'ST') AND (sLowerCase = 'sendboardinfo') THEN

			eMsgType					:= HermesMsgTypeSendBoardInfo;
			tyMsgType.bSendBoardInfo	:= TRUE;
			iSendBoardInfoFirstIdx		:= iHermesIdx;

		ELSIF (p_tyXMLTable.sTitle = 'ST') AND (sLowerCase = 'queryworkorderinfo') THEN

			eMsgType				    	:= HermesMsgTypeQueryWorkOrderInfo;
			tyMsgType.bQueryWorkOrderInfo	:= TRUE;
			iQueryWorkOrderInfoFirstIdx		:= iHermesIdx;

		ELSIF (p_tyXMLTable.sTitle = 'ST') AND (sLowerCase = 'sendworkorderinfo') THEN

			eMsgType				    	:= HermesMsgTypeSendWorkOrderInfo;
			tyMsgType.bSendWorkOrderInfo	:= TRUE;
			iSendWorkOrderInfoFirstIdx		:= iHermesIdx;
		ELSIF (p_tyXMLTable.sTitle = 'ST') AND (sLowerCase = 'command') THEN

			eMsgType						:= HermesMsgTypeCommand;
			tyMsgType.bCommand				:= TRUE;
			iCommandFirstIdx				:= iHermesIdx;
		ELSE

			CASE eMsgType OF
				HermesMsgTypeCheckAlive:
					fHermesParseCheckAlive(ADR(tyCheckAlive) , p_tyXMLTable , p_tyXMLTable1 , sLowerCase);

				HermesMsgTypeServiceDescription:
					fHermesParseServiceDescription(ADR(tyServiceDescription) , p_tyXMLTable , p_tyXMLTable1 , sLowerCase);

				HermesMsgTypeSServiceDescription:
					fHermesParseSServiceDescription(ADR(tySServiceDescription) , p_tyXMLTable , p_tyXMLTable1 , sLowerCase);

				HermesMsgTypeNotification:
					fHermesParseNotification(ADR(tyNotification) , p_tyXMLTable , p_tyXMLTable1 , sLowerCase);

				HermesMsgTypeBoardAvailable:
					fHermesParseBoardAvailable(ADR(tyBoardAvailable) , p_tyXMLTable , p_tyXMLTable1 , sLowerCase,ADR(iSubBoardCntr));

				HermesMsgTypeMachineReady:
					fHermesParseMachineReady(ADR(tyMachineReady) , p_tyXMLTable , p_tyXMLTable1 , sLowerCase);

				HermesMsgTypeStartTransport:
					fHermesParseStartTransport(ADR(tyStartTransport) , p_tyXMLTable , p_tyXMLTable1 , sLowerCase);

				HermesMsgTypeStopTransport:
					fHermesParseStopTransport(ADR(tyStopTransport) , p_tyXMLTable , p_tyXMLTable1 , sLowerCase);

				HermesMsgTypeTransportFinished:
					fHermesParseTransportFinished(ADR(tyTransportFinished) , p_tyXMLTable , p_tyXMLTable1 , sLowerCase);

				HermesMsgTypeSetConfiguration:
					fHermesParseSetConfiguration(ADR(tySetConfiguration) , p_tyXMLTable , p_tyXMLTable1 , sLowerCase , bUpstream := bSetUpstream , bDownstream := bSetDownstream);

				HermesMsgTypeCurrConfiguration:
					fHermesParseCurrentConfiguration(ADR(tyCurrentConfiguration) , p_tyXMLTable , p_tyXMLTable1 , sLowerCase , bUpstream := bCurrUpstream , bDownstream := bCurrDownstream);

				HermesMsgTypeBoardForecast:
					fHermesParseBoardForecast(ADR(tyBoardForecast) , p_tyXMLTable , p_tyXMLTable1 , sLowerCase);

				HermesMsgTypeBoardArrived:
					fHermesParseBoardArrived(ADR(tyBoardArrived) , p_tyXMLTable , p_tyXMLTable1 , sLowerCase);

				HermesMsgTypeBoardDeparted:
					fHermesParseBoardDeparted(ADR(tyBoardDeparted) , p_tyXMLTable , p_tyXMLTable1 , sLowerCase);

				HermesMsgTypeQueryBoardInfo:
					fHermesParseQueryBoardInfo(ADR(tyQueryBoardInfo) , p_tyXMLTable , p_tyXMLTable1 , sLowerCase);

				HermesMsgTypeSendBoardInfo:
					fHermesParseSendBoardInfo(ADR(tySendBoardInfo) , p_tyXMLTable , p_tyXMLTable1 , sLowerCase);

				HermesMsgTypeQueryWorkOrderInfo:
					fHermesParseQueryWorkOrderInfo(ADR(tyQueryWorkOrderInfo) , p_tyXMLTable , p_tyXMLTable1 , sLowerCase);

				HermesMsgTypeSendWorkOrderInfo:
					fHermesParseSendWorkOrderInfo(ADR(tySendWorkOrderInfo) , p_tyXMLTable , p_tyXMLTable1 , sLowerCase);

				HermesMsgTypeCommand:
					fHermesParseCommand(ADR(tyCommand) , p_tyXMLTable , p_tyXMLTable1 , sLowerCase);

			END_CASE

		END_IF

	END_FOR

END_FUNCTION_BLOCK
```

#### fHermesParseServiceDescription.st
```iecst
(* Hermes Parse XML Table Data For ServiceDescription *)
FUNCTION fHermesParseServiceDescription

	fHermesParseServiceDescription	:= TRUE;

	IF (tyXMLTableCurr.sTitle = 'AT') AND (sCurrValueLowerCase = 'laneid') THEN

		p_tyServiceDescription.tyAvl.bLaneId	:= TRUE;

		IF tyXMLTableNxt.sTitle = 'AV' THEN
			p_tyServiceDescription.tyData.iLaneId	:= STRING_TO_INT(tyXMLTableNxt.sValue);
		END_IF

	ELSIF (tyXMLTableCurr.sTitle = 'AT') AND (sCurrValueLowerCase = 'machineid') THEN

		p_tyServiceDescription.tyAvl.bMachineId	:= TRUE;

		IF tyXMLTableNxt.sTitle = 'AV' THEN
			p_tyServiceDescription.tyData.sMachineId	:= tyXMLTableNxt.sValue;
		END_IF

	ELSIF (tyXMLTableCurr.sTitle = 'AT') AND (sCurrValueLowerCase = 'interfaceid') THEN

		p_tyServiceDescription.tyAvl.bInterfaceId	:= TRUE;

		IF tyXMLTableNxt.sTitle = 'AV' THEN
			p_tyServiceDescription.tyData.sInterfaceId	:= tyXMLTableNxt.sValue;
		END_IF

	ELSIF (tyXMLTableCurr.sTitle = 'AT') AND (sCurrValueLowerCase = 'version') THEN

		p_tyServiceDescription.tyAvl.bVersion	:= TRUE;

		IF tyXMLTableNxt.sTitle = 'AV' THEN
			p_tyServiceDescription.tyData.sVersion	:= tyXMLTableNxt.sValue;
		END_IF

	ELSIF (tyXMLTableCurr.sTitle = 'ST') AND (sCurrValueLowerCase = 'supportedfeatures') THEN

		p_tyServiceDescription.tyAvl.bSupportedFeatures	:= TRUE;

	ELSIF (tyXMLTableCurr.sTitle = 'ST') AND (sCurrValueLowerCase = 'featureboardforecast') THEN

		p_tyServiceDescription.tyAvl.tySupportedFeatures.bFeatureBoardForecast	:= TRUE;
		p_tyServiceDescription.tyData.tySupportedFeatures.bFeatureBoardForecast	:= TRUE;

	ELSIF (tyXMLTableCurr.sTitle = 'ST') AND (sCurrValueLowerCase = 'featurecheckaliveresponse') THEN

		p_tyServiceDescription.tyAvl.tySupportedFeatures.bFeatureCheckAliveResponse		:= TRUE;
		p_tyServiceDescription.tyData.tySupportedFeatures.bFeatureCheckAliveResponse	:= TRUE;

	ELSIF (tyXMLTableCurr.sTitle = 'ST') AND (sCurrValueLowerCase = 'featurequeryboardinfo') THEN

		p_tyServiceDescription.tyAvl.tySupportedFeatures.bFeatureQueryBoardInfo		:= TRUE;
		p_tyServiceDescription.tyData.tySupportedFeatures.bFeatureQueryBoardInfo	:= TRUE;

	ELSIF (tyXMLTableCurr.sTitle = 'ST') AND (sCurrValueLowerCase = 'featuresendboardinfo') THEN

		p_tyServiceDescription.tyAvl.tySupportedFeatures.bFeatureSendBoardInfo	:= TRUE;
		p_tyServiceDescription.tyData.tySupportedFeatures.bFeatureSendBoardInfo	:= TRUE;

	ELSIF (tyXMLTableCurr.sTitle = 'ST') AND (sCurrValueLowerCase = 'featurecommand') THEN

		p_tyServiceDescription.tyAvl.tySupportedFeatures.bFeatureCommand	:= TRUE;
		p_tyServiceDescription.tyData.tySupportedFeatures.bFeatureCommand	:= TRUE;
	END_IF

END_FUNCTION
```

#### fHermesParseSServiceDescription.st
```iecst
(* Hermes Parse XML Table Data For Supervisory ServiceDescription *)
FUNCTION fHermesParseSServiceDescription

	fHermesParseSServiceDescription	:= TRUE;

    IF (tyXMLTableCurr.sTitle = 'AT') AND (sCurrValueLowerCase = 'systemid') THEN

		p_tySServiceDescription.tyAvl.bSystemId	:= TRUE;

		IF tyXMLTableNxt.sTitle = 'AV' THEN
			p_tySServiceDescription.tyData.sSystemId	:= tyXMLTableNxt.sValue;
		END_IF

	ELSIF (tyXMLTableCurr.sTitle = 'AT') AND (sCurrValueLowerCase = 'version') THEN

		p_tySServiceDescription.tyAvl.bVersion	:= TRUE;

		IF tyXMLTableNxt.sTitle = 'AV' THEN
			p_tySServiceDescription.tyData.sVersion	:= tyXMLTableNxt.sValue;
		END_IF

	ELSIF (tyXMLTableCurr.sTitle = 'ST') AND (sCurrValueLowerCase = 'supportedfeatures') THEN

		p_tySServiceDescription.tyAvl.bSupportedFeatures	:= TRUE;

	ELSIF (tyXMLTableCurr.sTitle = 'ST') AND (sCurrValueLowerCase = 'featureconfiguration') THEN

		p_tySServiceDescription.tyAvl.tySupportedFeatures.bFeatureConfiguration	:= TRUE;
		p_tySServiceDescription.tyData.tySupportedFeatures.bFeatureConfiguration	:= TRUE;

	ELSIF (tyXMLTableCurr.sTitle = 'ST') AND (sCurrValueLowerCase = 'featurecheckaliveresponse') THEN

		p_tySServiceDescription.tyAvl.tySupportedFeatures.bFeatureCheckAliveResponse		:= TRUE;
		p_tySServiceDescription.tyData.tySupportedFeatures.bFeatureCheckAliveResponse	:= TRUE;

	ELSIF (tyXMLTableCurr.sTitle = 'ST') AND (sCurrValueLowerCase = 'featureboardtracking') THEN

		p_tySServiceDescription.tyAvl.tySupportedFeatures.bFeatureBoardTracking		:= TRUE;
		p_tySServiceDescription.tyData.tySupportedFeatures.bFeatureBoardTracking	:= TRUE;

	ELSIF (tyXMLTableCurr.sTitle = 'ST') AND (sCurrValueLowerCase = 'featurequeryworkorderinfo') THEN

		p_tySServiceDescription.tyAvl.tySupportedFeatures.bFeatureQueryWorkOrderInfo	:= TRUE;
		p_tySServiceDescription.tyData.tySupportedFeatures.bFeatureQueryWorkOrderInfo	:= TRUE;

	ELSIF (tyXMLTableCurr.sTitle = 'ST') AND (sCurrValueLowerCase = 'featuresendworkorderinfo') THEN

		p_tySServiceDescription.tyAvl.tySupportedFeatures.bFeatureSendWorkOrderInfo	:= TRUE;
		p_tySServiceDescription.tyData.tySupportedFeatures.bFeatureSendWorkOrderInfo	:= TRUE;

	END_IF

END_FUNCTION
```

#### fHermesParseCheckAlive.st
```iecst
(* Hermes Parse XML Table Data For Check Alive *)
FUNCTION fHermesParseCheckAlive

	fHermesParseCheckAlive	:= TRUE;

	IF (tyXMLTableCurr.sTitle = 'AT') AND (sCurrValueLowerCase = 'type') THEN

		p_tyCheckAlive.tyAvl.bType	:= TRUE;

		IF tyXMLTableNxt.sTitle = 'AV' THEN
			IF tyXMLTableNxt.sValue = '1' THEN
				p_tyCheckAlive.tyData.eType	:= HermesCheckAliveTypePing;
			ELSIF tyXMLTableNxt.sValue = '2' THEN
				p_tyCheckAlive.tyData.eType	:= HermesCheckAliveTypePong;
			ELSE
				p_tyCheckAlive.tyData.eType	:= HermesCheckAliveTypeUnknown;
			END_IF
		END_IF

	ELSIF (tyXMLTableCurr.sTitle = 'AT') AND (sCurrValueLowerCase = 'id') THEN

		p_tyCheckAlive.tyAvl.bId	:= TRUE;

		IF tyXMLTableNxt.sTitle = 'AV' THEN
			p_tyCheckAlive.tyData.sId	:= tyXMLTableNxt.sValue;
		END_IF

	END_IF

END_FUNCTION
```

#### fHermesParseNotification.st
```iecst
(* Hermes Parse XML Table Data For Notification *)
FUNCTION fHermesParseNotification

	fHermesParseNotification	:= TRUE;

	IF (tyXMLTableCurr.sTitle = 'AT') AND (sCurrValueLowerCase = 'notificationcode') THEN

		p_tyNotification.tyAvl.bNotificationCode	:= TRUE;

		IF tyXMLTableNxt.sTitle = 'AV' THEN
			p_tyNotification.tyData.iNotificationCode	:= STRING_TO_INT(tyXMLTableNxt.sValue);
		END_IF

	ELSIF (tyXMLTableCurr.sTitle = 'AT') AND (sCurrValueLowerCase = 'severity') THEN

		p_tyNotification.tyAvl.bSeverity	:= TRUE;

		IF tyXMLTableNxt.sTitle = 'AV' THEN
			IF tyXMLTableNxt.sValue = '1' THEN
				p_tyNotification.tyData.eSeverity	:= HermesSeverityFatalError;
			ELSIF tyXMLTableNxt.sValue = '2' THEN
				p_tyNotification.tyData.eSeverity	:= HermesSeverityError;
			ELSIF tyXMLTableNxt.sValue = '3' THEN
				p_tyNotification.tyData.eSeverity	:= HermesSeverityWarning;
			ELSE
				p_tyNotification.tyData.eSeverity	:= HermesSeverityInfo;
			END_IF
		END_IF

	ELSIF (tyXMLTableCurr.sTitle = 'AT') AND (sCurrValueLowerCase = 'description') THEN

		p_tyNotification.tyAvl.bDescription	:= TRUE;

		IF tyXMLTableNxt.sTitle = 'AV' THEN
			p_tyNotification.tyData.sDescription	:= tyXMLTableNxt.sValue;
		END_IF

	END_IF

END_FUNCTION
```
